gfCNCPoint3[3648] = {X 36.5946, Y 43.2362, Z -3.8333, A 0.000, B 0.000, C 0.000 }
gfCNCPoint3[3649] = {X 36.9340, Y 42.3177, Z -3.8333, A 0.000, B 0.000, C 0.000 }
gfCNCPoint3[3650] = {X 37.4786, Y 41.5040, Z -3.8333, A 0.000, B 0.000, C 0.000 }
gfCNCPoint3[3651] = {X 38.1984, Y 40.8401, Z -3.8333, A 0.000, B 0.000, C 0.000 }
gfCNCPoint3[3652] = {X 39.0535, Y 40.3629, Z -3.8333, A 0.000, B 0.000, C 0.000 }
gfCNCPoint3[3653] = {X 39.6603, Y 38.9339, Z -3.8333, A 0.000, B 0.000, C 0.000 }
gfCNCPoint3[3654] = {X 40.2151, Y 37.4838, Z -3.8333, A 0.000, B 0.000, C 0.000 }
gfCNCPoint3[3655] = {X 43.7985, Y 27.8628, Z -3.8333, A 0.000, B 0.000, C 0.000 }
gfCNCPoint3[3656] = {X 40.0500, Y 26.4667, Z -3.8333, A 0.000, B 0.000, C 0.000 }
gfCNCPoint3[3657] = {X 43.8734, Y 27.8908, Z -3.8333, A 0.000, B 0.000, C 0.000 }
gfCNCPoint3[3658] = {X 48.5582, Y 15.3126, Z -3.8333, A 0.000, B 0.000, C 0.000 }
gfCNCPoint3[3659] = {X 48.1610, Y 14.6012, Z -3.8333, A 0.000, B 0.000, C 0.000 }
gfCNCPoint3[3660] = {X 47.9131, Y 13.8250, Z -3.8333, A 0.000, B 0.000, C 0.000 }
gfCNCPoint3[3661] = {X 47.8244, Y 13.0151, Z -3.8333, A 0.000, B 0.000, C 0.000 }
gfCNCPoint3[3662] = {X 47.8242, Y 12.1868, Z -3.8333, A 0.000, B 0.000, C 0.000 }
gfCNCPoint3[3663] = {X 47.9265, Y 11.2789, Z -3.8333, A 0.000, B 0.000, C 0.000 }
gfCNCPoint3[3664] = {X 48.2283, Y 10.4166, Z -3.8333, A 0.000, B 0.000, C 0.000 }
gfCNCPoint3[3665] = {X 48.7144, Y 9.6430, Z -3.8333, A 0.000, B 0.000, C 0.000 }
gfCNCPoint3[3666] = {X 49.3604, Y 8.9969, Z -3.8333, A 0.000, B 0.000, C 0.000 }
gfCNCPoint3[3667] = {X 50.1340, Y 8.5109, Z -3.8333, A 0.000, B 0.000, C 0.000 }
gfCNCPoint3[3668] = {X 50.9963, Y 8.2091, Z -3.8333, A 0.000, B 0.000, C 0.000 }
gfCNCPoint3[3669] = {X 51.9042, Y 8.1068, Z -3.8333, A 0.000, B 0.000, C 0.000 }
gfCNCPoint3[3670] = {X 59.6221, Y 8.1068, Z -3.8333, A 0.000, B 0.000, C 0.000 }
gfCNCPoint3[3671] = {X 60.5300, Y 8.2091, Z -3.8333, A 0.000, B 0.000, C 0.000 }
gfCNCPoint3[3672] = {X 61.3924, Y 8.5109, Z -3.8333, A 0.000, B 0.000, C 0.000 }
gfCNCPoint3[3673] = {X 62.1660, Y 8.9969, Z -3.8333, A 0.000, B 0.000, C 0.000 }
gfCNCPoint3[3674] = {X 62.8120, Y 9.6430, Z -3.8333, A 0.000, B 0.000, C 0.000 }
gfCNCPoint3[3675] = {X 63.2981, Y 10.4166, Z -3.8333, A 0.000, B 0.000, C 0.000 }
gfCNCPoint3[3676] = {X 63.5998, Y 11.2789, Z -3.8333, A 0.000, B 0.000, C 0.000 }
gfCNCPoint3[3677] = {X 63.7021, Y 12.1868, Z -3.8333, A 0.000, B 0.000, C 0.000 }
gfCNCPoint3[3678] = {X 63.7021, Y 12.9781, Z -3.8333, A 0.000, B 0.000, C 0.000 }
gfCNCPoint3[3679] = {X 63.6148, Y 13.8178, Z -3.8333, A 0.000, B 0.000, C 0.000 }
gfCNCPoint3[3680] = {X 63.3565, Y 14.6215, Z -3.8333, A 0.000, B 0.000, C 0.000 }
gfCNCPoint3[3681] = {X 62.9383, Y 15.3549, Z -3.8333, A 0.000, B 0.000, C 0.000 }
gfCNCPoint3[3682] = {X 63.2010, Y 16.0481, Z -3.8333, A 0.000, B 0.000, C 0.000 }
gfCNCPoint3[3683] = {X 66.0153, Y 23.5156, Z -3.8333, A 0.000, B 0.000, C 0.000 }
gfCNCPoint3[3684] = {X 71.9853, Y 39.5865, Z -3.8333, A 0.000, B 0.000, C 0.000 }
gfCNCPoint3[3685] = {X 72.3281, Y 40.4487, Z -3.8333, A 0.000, B 0.000, C 0.000 }
gfCNCPoint3[3686] = {X 73.1522, Y 40.9150, Z -3.8333, A 0.000, B 0.000, C 0.000 }
gfCNCPoint3[3687] = {X 73.8466, Y 41.5587, Z -3.8333, A 0.000, B 0.000, C 0.000 }
gfCNCPoint3[3688] = {X 74.3739, Y 42.3451, Z -3.8333, A 0.000, B 0.000, C 0.000 }
gfCNCPoint3[3689] = {X 74.7058, Y 43.2319, Z -3.8333, A 0.000, B 0.000, C 0.000 }
gfCNCPoint3[3690] = {X 74.8243, Y 44.1714, Z -3.8333, A 0.000, B 0.000, C 0.000 }
gfCNCPoint3[3691] = {X 74.8245, Y 45.0000, Z -3.8333, A 0.000, B 0.000, C 0.000 }
gfCNCPoint3[3692] = {X 74.7222, Y 45.9079, Z -3.8333, A 0.000, B 0.000, C 0.000 }
gfCNCPoint3[3693] = {X 74.4204, Y 46.7702, Z -3.8333, A 0.000, B 0.000, C 0.000 }
gfCNCPoint3[3694] = {X 73.9343, Y 47.5438, Z -3.8333, A 0.000, B 0.000, C 0.000 }
gfCNCPoint3[3695] = {X 73.2883, Y 48.1899, Z -3.8333, A 0.000, B 0.000, C 0.000 }
gfCNCPoint3[3696] = {X 72.5147, Y 48.6760, Z -3.8333, A 0.000, B 0.000, C 0.000 }
gfCNCPoint3[3697] = {X 71.6523, Y 48.9777, Z -3.8333, A 0.000, B 0.000, C 0.000 }
gfCNCPoint3[3698] = {X 70.7445, Y 49.0800, Z -3.8333, A 0.000, B 0.000, C 0.000 }
gfCNCPoint3[3699] = {X 64.1851, Y 49.0800, Z -3.8333, A 0.000, B 0.000, C 0.000 }
gfCNCPoint3[3700] = {X 63.2772, Y 48.9777, Z -3.8333, A 0.000, B 0.000, C 0.000 }
gfCNCPoint3[3701] = {X 62.4149, Y 48.6760, Z -3.8333, A 0.000, B 0.000, C 0.000 }
gfCNCPoint3[3702] = {X 61.6413, Y 48.1899, Z -3.8333, A 0.000, B 0.000, C 0.000 }
gfCNCPoint3[3703] = {X 60.9953, Y 47.5438, Z -3.8333, A 0.000, B 0.000, C 0.000 }
gfCNCPoint3[3704] = {X 60.5092, Y 46.7702, Z -3.8333, A 0.000, B 0.000, C 0.000 }
gfCNCPoint3[3705] = {X 60.2074, Y 45.9079, Z -3.8333, A 0.000, B 0.000, C 0.000 }
gfCNCPoint3[3706] = {X 60.1051, Y 45.0000, Z -3.8333, A 0.000, B 0.000, C 0.000 }
gfCNCPoint3[3707] = {X 60.1051, Y 44.2086, Z -3.8333, A 0.000, B 0.000, C 0.000 }
gfCNCPoint3[3708] = {X 60.1954, Y 43.3580, Z -3.8333, A 0.000, B 0.000, C 0.000 }
gfCNCPoint3[3709] = {X 60.4611, Y 42.5449, Z -3.8333, A 0.000, B 0.000, C 0.000 }
gfCNCPoint3[3710] = {X 60.8905, Y 41.8050, Z -3.8333, A 0.000, B 0.000, C 0.000 }
gfCNCPoint3[3711] = {X 60.1748, Y 39.8492, Z -3.8333, A 0.000, B 0.000, C 0.000 }
gfCNCPoint3[3712] = {X 51.9103, Y 39.8492, Z -3.8333, A 0.000, B 0.000, C 0.000 }
gfCNCPoint3[3713] = {X 51.0690, Y 42.1092, Z -3.8333, A 0.000, B 0.000, C 0.000 }
gfCNCPoint3[3714] = {X 51.1306, Y 42.2115, Z -3.8333, A 0.000, B 0.000, C 0.000 }
gfCNCPoint3[3715] = {X 51.4141, Y 42.8332, Z -3.8333, A 0.000, B 0.000, C 0.000 }
gfCNCPoint3[3716] = {X 51.5898, Y 43.4936, Z -3.8333, A 0.000, B 0.000, C 0.000 }
gfCNCPoint3[3717] = {X 51.6528, Y 44.1740, Z -3.8333, A 0.000, B 0.000, C 0.000 }
gfCNCPoint3[3718] = {X 51.6529, Y 45.0000, Z -3.8333, A 0.000, B 0.000, C 0.000 }
gfCNCPoint3[3719] = {X 51.5506, Y 45.9079, Z -3.8333, A 0.000, B 0.000, C 0.000 }
gfCNCPoint3[3720] = {X 51.2489, Y 46.7702, Z -3.8333, A 0.000, B 0.000, C 0.000 }
gfCNCPoint3[3721] = {X 50.7628, Y 47.5438, Z -3.8333, A 0.000, B 0.000, C 0.000 }
gfCNCPoint3[3722] = {X 50.1168, Y 48.1899, Z -3.8333, A 0.000, B 0.000, C 0.000 }
gfCNCPoint3[3723] = {X 49.3432, Y 48.6760, Z -3.8333, A 0.000, B 0.000, C 0.000 }
gfCNCPoint3[3724] = {X 48.4808, Y 48.9777, Z -3.8333, A 0.000, B 0.000, C 0.000 }
gfCNCPoint3[3725] = {X 47.5729, Y 49.0800, Z -3.8333, A 0.000, B 0.000, C 0.000 }
gfCNCPoint3[3726] = {X 40.6393, Y 49.0800, Z -3.8333, A 0.000, B 0.000, C 0.000 }
gfCNCPoint3[3727] = {X 39.7314, Y 48.9777, Z -3.8333, A 0.000, B 0.000, C 0.000 }
gfCNCPoint3[3728] = {X 38.8691, Y 48.6760, Z -3.8333, A 0.000, B 0.000, C 0.000 }
gfCNCPoint3[3729] = {X 38.0955, Y 48.1899, Z -3.8333, A 0.000, B 0.000, C 0.000 }
gfCNCPoint3[3730] = {X 37.4494, Y 47.5438, Z -3.8333, A 0.000, B 0.000, C 0.000 }
gfCNCPoint3[3731] = {X 36.9633, Y 46.7702, Z -3.8333, A 0.000, B 0.000, C 0.000 }
gfCNCPoint3[3732] = {X 36.6616, Y 45.9079, Z -3.8333, A 0.000, B 0.000, C 0.000 }
gfCNCPoint3[3733] = {X 36.5593, Y 45.0000, Z -3.8333, A 0.000, B 0.000, C 0.000 }
gfCNCPoint3[3734] = {X 36.5593, Y 44.2086, Z -3.8333, A 0.000, B 0.000, C 0.000 }
gfCNCPoint3[3735] = {X 36.6737, Y 43.2478, Z -3.8333, A 0.000, B 0.000, C 0.000 }
gfCNCPoint3[3736] = {X 37.0110, Y 42.3409, Z -3.8333, A 0.000, B 0.000, C 0.000 }
gfCNCPoint3[3737] = {X 37.5522, Y 41.5388, Z -3.8333, A 0.000, B 0.000, C 0.000 }
gfCNCPoint3[3738] = {X 38.2670, Y 40.8866, Z -3.8333, A 0.000, B 0.000, C 0.000 }
gfCNCPoint3[3739] = {X 39.1152, Y 40.4209, Z -3.8333, A 0.000, B 0.000, C 0.000 }
gfCNCPoint3[3740] = {X 39.1265, Y 40.3955, Z -3.8333, A 0.000, B 0.000, C 0.000 }
gfCNCPoint3[3741] = {X 39.7345, Y 38.9638, Z -3.8333, A 0.000, B 0.000, C 0.000 }
gfCNCPoint3[3742] = {X 40.2904, Y 37.5110, Z -3.8333, A 0.000, B 0.000, C 0.000 }
gfCNCPoint3[3743] = {X 43.8734, Y 27.8908, Z -3.8333, A 0.000, B 0.000, C 0.000 }
gfCNCPoint3[3744] = {X 40.1250, Y 26.4946, Z -3.8333, A 0.000, B 0.000, C 0.000 }
gfCNCPoint3[3745] = {X 43.9484, Y 27.9187, Z -3.8333, A 0.000, B 0.000, C 0.000 }
gfCNCPoint3[3746] = {X 48.6479, Y 15.3010, Z -3.8333, A 0.000, B 0.000, C 0.000 }
gfCNCPoint3[3747] = {X 48.2407, Y 14.5838, Z -3.8333, A 0.000, B 0.000, C 0.000 }
gfCNCPoint3[3748] = {X 47.9892, Y 13.7983, Z -3.8333, A 0.000, B 0.000, C 0.000 }
gfCNCPoint3[3749] = {X 47.9042, Y 12.9779, Z -3.8333, A 0.000, B 0.000, C 0.000 }
gfCNCPoint3[3750] = {X 47.9042, Y 12.1868, Z -3.8333, A 0.000, B 0.000, C 0.000 }
gfCNCPoint3[3751] = {X 48.0045, Y 11.2967, Z -3.8333, A 0.000, B 0.000, C 0.000 }
gfCNCPoint3[3752] = {X 48.3003, Y 10.4513, Z -3.8333, A 0.000, B 0.000, C 0.000 }
gfCNCPoint3[3753] = {X 48.7769, Y 9.6929, Z -3.8333, A 0.000, B 0.000, C 0.000 }
gfCNCPoint3[3754] = {X 49.4103, Y 9.0595, Z -3.8333, A 0.000, B 0.000, C 0.000 }
gfCNCPoint3[3755] = {X 50.1687, Y 8.5829, Z -3.8333, A 0.000, B 0.000, C 0.000 }
gfCNCPoint3[3756] = {X 51.0141, Y 8.2871, Z -3.8333, A 0.000, B 0.000, C 0.000 }
gfCNCPoint3[3757] = {X 51.9042, Y 8.1868, Z -3.8333, A 0.000, B 0.000, C 0.000 }
gfCNCPoint3[3758] = {X 59.6221, Y 8.1868, Z -3.8333, A 0.000, B 0.000, C 0.000 }
gfCNCPoint3[3759] = {X 60.5122, Y 8.2871, Z -3.8333, A 0.000, B 0.000, C 0.000 }
gfCNCPoint3[3760] = {X 61.3577, Y 8.5829, Z -3.8333, A 0.000, B 0.000, C 0.000 }
gfCNCPoint3[3761] = {X 62.1161, Y 9.0595, Z -3.8333, A 0.000, B 0.000, C 0.000 }
gfCNCPoint3[3762] = {X 62.7495, Y 9.6929, Z -3.8333, A 0.000, B 0.000, C 0.000 }
gfCNCPoint3[3763] = {X 63.2260, Y 10.4513, Z -3.8333, A 0.000, B 0.000, C 0.000 }
gfCNCPoint3[3764] = {X 63.5218, Y 11.2967, Z -3.8333, A 0.000, B 0.000, C 0.000 }
gfCNCPoint3[3765] = {X 63.6221, Y 12.1868, Z -3.8333, A 0.000, B 0.000, C 0.000 }
gfCNCPoint3[3766] = {X 63.6219, Y 13.0192, Z -3.8333, A 0.000, B 0.000, C 0.000 }
gfCNCPoint3[3767] = {X 63.5277, Y 13.8420, Z -3.8333, A 0.000, B 0.000, C 0.000 }
gfCNCPoint3[3768] = {X 63.2660, Y 14.6278, Z -3.8333, A 0.000, B 0.000, C 0.000 }
gfCNCPoint3[3769] = {X 62.8482, Y 15.3429, Z -3.8333, A 0.000, B 0.000, C 0.000 }
gfCNCPoint3[3770] = {X 63.1261, Y 16.0764, Z -3.8333, A 0.000, B 0.000, C 0.000 }
gfCNCPoint3[3771] = {X 65.9404, Y 23.5436, Z -3.8333, A 0.000, B 0.000, C 0.000 }
gfCNCPoint3[3772] = {X 71.9107, Y 39.6152, Z -3.8333, A 0.000, B 0.000, C 0.000 }
gfCNCPoint3[3773] = {X 72.2611, Y 40.4966, Z -3.8333, A 0.000, B 0.000, C 0.000 }
gfCNCPoint3[3774] = {X 72.2790, Y 40.5149, Z -3.8333, A 0.000, B 0.000, C 0.000 }
gfCNCPoint3[3775] = {X 72.3450, Y 40.5429, Z -3.8333, A 0.000, B 0.000, C 0.000 }
gfCNCPoint3[3776] = {X 72.4104, Y 40.5722, Z -3.8333, A 0.000, B 0.000, C 0.000 }
gfCNCPoint3[3777] = {X 73.1900, Y 41.0435, Z -3.8333, A 0.000, B 0.000, C 0.000 }
gfCNCPoint3[3778] = {X 73.8428, Y 41.6790, Z -3.8333, A 0.000, B 0.000, C 0.000 }
gfCNCPoint3[3779] = {X 74.3349, Y 42.4457, Z -3.8333, A 0.000, B 0.000, C 0.000 }
gfCNCPoint3[3780] = {X 74.6407, Y 43.3038, Z -3.8333, A 0.000, B 0.000, C 0.000 }
gfCNCPoint3[3781] = {X 74.7445, Y 44.2089, Z -3.8333, A 0.000, B 0.000, C 0.000 }
gfCNCPoint3[3782] = {X 74.7445, Y 45.0000, Z -3.8333, A 0.000, B 0.000, C 0.000 }
gfCNCPoint3[3783] = {X 74.6442, Y 45.8901, Z -3.8333, A 0.000, B 0.000, C 0.000 }
gfCNCPoint3[3784] = {X 74.3483, Y 46.7355, Z -3.8333, A 0.000, B 0.000, C 0.000 }
gfCNCPoint3[3785] = {X 73.8718, Y 47.4940, Z -3.8333, A 0.000, B 0.000, C 0.000 }
gfCNCPoint3[3786] = {X 73.2384, Y 48.1273, Z -3.8333, A 0.000, B 0.000, C 0.000 }
gfCNCPoint3[3787] = {X 72.4800, Y 48.6039, Z -3.8333, A 0.000, B 0.000, C 0.000 }
gfCNCPoint3[3788] = {X 71.6345, Y 48.8997, Z -3.8333, A 0.000, B 0.000, C 0.000 }
gfCNCPoint3[3789] = {X 70.7445, Y 49.0000, Z -3.8333, A 0.000, B 0.000, C 0.000 }
gfCNCPoint3[3790] = {X 64.1851, Y 49.0000, Z -3.8333, A 0.000, B 0.000, C 0.000 }
gfCNCPoint3[3791] = {X 63.2951, Y 48.8997, Z -3.8333, A 0.000, B 0.000, C 0.000 }
gfCNCPoint3[3792] = {X 62.4496, Y 48.6039, Z -3.8333, A 0.000, B 0.000, C 0.000 }
gfCNCPoint3[3793] = {X 61.6912, Y 48.1273, Z -3.8333, A 0.000, B 0.000, C 0.000 }
gfCNCPoint3[3794] = {X 61.0578, Y 47.4940, Z -3.8333, A 0.000, B 0.000, C 0.000 }
gfCNCPoint3[3795] = {X 60.5813, Y 46.7355, Z -3.8333, A 0.000, B 0.000, C 0.000 }
gfCNCPoint3[3796] = {X 60.2854, Y 45.8901, Z -3.8333, A 0.000, B 0.000, C 0.000 }
gfCNCPoint3[3797] = {X 60.1851, Y 45.0000, Z -3.8333, A 0.000, B 0.000, C 0.000 }
gfCNCPoint3[3798] = {X 60.1855, Y 44.1538, Z -3.8333, A 0.000, B 0.000, C 0.000 }
gfCNCPoint3[3799] = {X 60.2746, Y 43.3674, Z -3.8333, A 0.000, B 0.000, C 0.000 }
gfCNCPoint3[3800] = {X 60.5168, Y 42.6140, Z -3.8333, A 0.000, B 0.000, C 0.000 }
gfCNCPoint3[3801] = {X 60.9025, Y 41.9231, Z -3.8333, A 0.000, B 0.000, C 0.000 }
gfCNCPoint3[3802] = {X 60.9805, Y 41.8180, Z -3.8333, A 0.000, B 0.000, C 0.000 }
gfCNCPoint3[3803] = {X 60.2307, Y 39.7692, Z -3.8333, A 0.000, B 0.000, C 0.000 }
gfCNCPoint3[3804] = {X 51.8423, Y 39.7692, Z -3.8333, A 0.000, B 0.000, C 0.000 }
gfCNCPoint3[3805] = {X 51.8423, Y 39.8027, Z -3.8333, A 0.000, B 0.000, C 0.000 }
gfCNCPoint3[3806] = {X 50.9806, Y 42.1175, Z -3.8333, A 0.000, B 0.000, C 0.000 }
gfCNCPoint3[3807] = {X 51.0724, Y 42.2713, Z -3.8333, A 0.000, B 0.000, C 0.000 }
gfCNCPoint3[3808] = {X 51.3478, Y 42.8858, Z -3.8333, A 0.000, B 0.000, C 0.000 }
gfCNCPoint3[3809] = {X 51.5163, Y 43.5378, Z -3.8333, A 0.000, B 0.000, C 0.000 }
gfCNCPoint3[3810] = {X 51.5729, Y 44.2089, Z -3.8333, A 0.000, B 0.000, C 0.000 }
gfCNCPoint3[3811] = {X 51.5729, Y 45.0000, Z -3.8333, A 0.000, B 0.000, C 0.000 }
gfCNCPoint3[3812] = {X 51.4726, Y 45.8901, Z -3.8333, A 0.000, B 0.000, C 0.000 }
gfCNCPoint3[3813] = {X 51.1768, Y 46.7355, Z -3.8333, A 0.000, B 0.000, C 0.000 }
gfCNCPoint3[3814] = {X 50.7003, Y 47.4940, Z -3.8333, A 0.000, B 0.000, C 0.000 }
gfCNCPoint3[3815] = {X 50.0669, Y 48.1273, Z -3.8333, A 0.000, B 0.000, C 0.000 }
gfCNCPoint3[3816] = {X 49.3085, Y 48.6039, Z -3.8333, A 0.000, B 0.000, C 0.000 }
gfCNCPoint3[3817] = {X 48.4630, Y 48.8997, Z -3.8333, A 0.000, B 0.000, C 0.000 }
gfCNCPoint3[3818] = {X 47.5729, Y 49.0000, Z -3.8333, A 0.000, B 0.000, C 0.000 }
gfCNCPoint3[3819] = {X 40.6393, Y 49.0000, Z -3.8333, A 0.000, B 0.000, C 0.000 }
gfCNCPoint3[3820] = {X 39.7492, Y 48.8997, Z -3.8333, A 0.000, B 0.000, C 0.000 }
gfCNCPoint3[3821] = {X 38.9038, Y 48.6039, Z -3.8333, A 0.000, B 0.000, C 0.000 }
gfCNCPoint3[3822] = {X 38.1453, Y 48.1273, Z -3.8333, A 0.000, B 0.000, C 0.000 }
gfCNCPoint3[3823] = {X 37.5120, Y 47.4940, Z -3.8333, A 0.000, B 0.000, C 0.000 }
gfCNCPoint3[3824] = {X 37.0354, Y 46.7355, Z -3.8333, A 0.000, B 0.000, C 0.000 }
gfCNCPoint3[3825] = {X 36.7396, Y 45.8901, Z -3.8333, A 0.000, B 0.000, C 0.000 }
gfCNCPoint3[3826] = {X 36.6393, Y 45.0000, Z -3.8333, A 0.000, B 0.000, C 0.000 }
gfCNCPoint3[3827] = {X 36.6397, Y 44.1538, Z -3.8333, A 0.000, B 0.000, C 0.000 }
gfCNCPoint3[3828] = {X 36.7564, Y 43.2482, Z -3.8333, A 0.000, B 0.000, C 0.000 }
gfCNCPoint3[3829] = {X 37.0754, Y 42.3926, Z -3.8333, A 0.000, B 0.000, C 0.000 }
gfCNCPoint3[3830] = {X 37.5801, Y 41.6317, Z -3.8333, A 0.000, B 0.000, C 0.000 }
gfCNCPoint3[3831] = {X 38.2442, Y 41.0051, Z -3.8333, A 0.000, B 0.000, C 0.000 }
gfCNCPoint3[3832] = {X 39.0332, Y 40.5454, Z -3.8333, A 0.000, B 0.000, C 0.000 }
gfCNCPoint3[3833] = {X 39.0861, Y 40.5226, Z -3.8333, A 0.000, B 0.000, C 0.000 }
gfCNCPoint3[3834] = {X 39.1394, Y 40.5006, Z -3.8333, A 0.000, B 0.000, C 0.000 }
gfCNCPoint3[3835] = {X 39.1684, Y 40.4818, Z -3.8333, A 0.000, B 0.000, C 0.000 }
gfCNCPoint3[3836] = {X 39.1882, Y 40.4536, Z -3.8333, A 0.000, B 0.000, C 0.000 }
gfCNCPoint3[3837] = {X 39.2132, Y 40.3974, Z -3.8333, A 0.000, B 0.000, C 0.000 }
gfCNCPoint3[3838] = {X 39.2382, Y 40.3412, Z -3.8333, A 0.000, B 0.000, C 0.000 }
gfCNCPoint3[3839] = {X 39.8265, Y 38.9496, Z -3.8333, A 0.000, B 0.000, C 0.000 }
gfCNCPoint3[3840] = {X 40.3656, Y 37.5383, Z -3.8333, A 0.000, B 0.000, C 0.000 }
gfCNCPoint3[3841] = {X 43.9484, Y 27.9187, Z -3.8333, A 0.000, B 0.000, C 0.000 }
gfCNCPoint3[3842] = {X 40.1250, Y 26.4946, Z -3.8333, A 0.000, B 0.000, C 0.000 }
gfCNCPoint3[3843] = {X 40.1250, Y 26.4946, Z -0.8333, A 0.000, B 0.000, C 0.000 }
gfCNCPoint3[3844] = {X 40.1250, Y 26.4946, Z 11.0000, A 0.000, B 0.000, C 0.000 }
gfCNCPoint3[3845] = {X 79.0230, Y 28.5918, Z 11.0000, A 0.000, B 0.000, C 0.000 }
gfCNCPoint3[3846] = {X 79.0230, Y 28.5918, Z -0.8333, A 0.000, B 0.000, C 0.000 }
gfCNCPoint3[3847] = {X 79.0230, Y 28.5918, Z -3.8333, A 0.000, B 0.000, C 0.000 }
gfCNCPoint3[3848] = {X 83.1030, Y 28.5918, Z -3.8333, A 0.000, B 0.000, C 0.000 }
gfCNCPoint3[3849] = {X 83.1028, Y 16.2743, Z -3.8333, A 0.000, B 0.000, C 0.000 }
gfCNCPoint3[3850] = {X 82.4642, Y 15.6032, Z -3.8333, A 0.000, B 0.000, C 0.000 }
gfCNCPoint3[3851] = {X 81.9834, Y 14.8113, Z -3.8333, A 0.000, B 0.000, C 0.000 }
gfCNCPoint3[3852] = {X 81.6824, Y 13.9352, Z -3.8333, A 0.000, B 0.000, C 0.000 }
gfCNCPoint3[3853] = {X 81.5752, Y 13.0150, Z -3.8333, A 0.000, B 0.000, C 0.000 }
gfCNCPoint3[3854] = {X 81.5751, Y 12.1868, Z -3.8333, A 0.000, B 0.000, C 0.000 }
gfCNCPoint3[3855] = {X 81.6834, Y 11.2255, Z -3.8333, A 0.000, B 0.000, C 0.000 }
gfCNCPoint3[3856] = {X 82.0029, Y 10.3124, Z -3.8333, A 0.000, B 0.000, C 0.000 }
gfCNCPoint3[3857] = {X 82.5176, Y 9.4933, Z -3.8333, A 0.000, B 0.000, C 0.000 }
gfCNCPoint3[3858] = {X 83.2016, Y 8.8093, Z -3.8333, A 0.000, B 0.000, C 0.000 }
gfCNCPoint3[3859] = {X 84.0207, Y 8.2946, Z -3.8333, A 0.000, B 0.000, C 0.000 }
gfCNCPoint3[3860] = {X 84.9338, Y 7.9751, Z -3.8333, A 0.000, B 0.000, C 0.000 }
gfCNCPoint3[3861] = {X 85.8951, Y 7.8668, Z -3.8333, A 0.000, B 0.000, C 0.000 }
gfCNCPoint3[3862] = {X 94.0497, Y 7.8668, Z -3.8333, A 0.000, B 0.000, C 0.000 }
gfCNCPoint3[3863] = {X 95.0110, Y 7.9751, Z -3.8333, A 0.000, B 0.000, C 0.000 }
gfCNCPoint3[3864] = {X 95.9240, Y 8.2946, Z -3.8333, A 0.000, B 0.000, C 0.000 }
gfCNCPoint3[3865] = {X 96.7431, Y 8.8093, Z -3.8333, A 0.000, B 0.000, C 0.000 }
gfCNCPoint3[3866] = {X 97.4272, Y 9.4933, Z -3.8333, A 0.000, B 0.000, C 0.000 }
gfCNCPoint3[3867] = {X 97.9419, Y 10.3124, Z -3.8333, A 0.000, B 0.000, C 0.000 }
gfCNCPoint3[3868] = {X 98.2614, Y 11.2255, Z -3.8333, A 0.000, B 0.000, C 0.000 }
gfCNCPoint3[3869] = {X 98.3697, Y 12.1868, Z -3.8333, A 0.000, B 0.000, C 0.000 }
gfCNCPoint3[3870] = {X 98.3697, Y 12.9782, Z -3.8333, A 0.000, B 0.000, C 0.000 }
gfCNCPoint3[3871] = {X 98.2967, Y 13.7681, Z -3.8333, A 0.000, B 0.000, C 0.000 }
gfCNCPoint3[3872] = {X 98.0804, Y 14.5314, Z -3.8333, A 0.000, B 0.000, C 0.000 }
gfCNCPoint3[3873] = {X 97.7283, Y 15.2423, Z -3.8333, A 0.000, B 0.000, C 0.000 }
gfCNCPoint3[3874] = {X 101.8779, Y 25.5293, Z -3.8333, A 0.000, B 0.000, C 0.000 }
gfCNCPoint3[3875] = {X 106.0166, Y 15.2216, Z -3.8333, A 0.000, B 0.000, C 0.000 }
gfCNCPoint3[3876] = {X 105.6762, Y 14.5287, Z -3.8333, A 0.000, B 0.000, C 0.000 }
gfCNCPoint3[3877] = {X 105.4645, Y 13.7862, Z -3.8333, A 0.000, B 0.000, C 0.000 }
gfCNCPoint3[3878] = {X 105.3885, Y 13.0179, Z -3.8333, A 0.000, B 0.000, C 0.000 }
gfCNCPoint3[3879] = {X 105.3883, Y 12.1868, Z -3.8333, A 0.000, B 0.000, C 0.000 }
gfCNCPoint3[3880] = {X 105.4966, Y 11.2255, Z -3.8333, A 0.000, B 0.000, C 0.000 }
gfCNCPoint3[3881] = {X 105.8161, Y 10.3124, Z -3.8333, A 0.000, B 0.000, C 0.000 }
gfCNCPoint3[3882] = {X 106.3308, Y 9.4933, Z -3.8333, A 0.000, B 0.000, C 0.000 }
gfCNCPoint3[3883] = {X 107.0148, Y 8.8093, Z -3.8333, A 0.000, B 0.000, C 0.000 }
gfCNCPoint3[3884] = {X 107.8339, Y 8.2946, Z -3.8333, A 0.000, B 0.000, C 0.000 }
gfCNCPoint3[3885] = {X 108.7470, Y 7.9751, Z -3.8333, A 0.000, B 0.000, C 0.000 }
gfCNCPoint3[3886] = {X 109.7083, Y 7.8668, Z -3.8333, A 0.000, B 0.000, C 0.000 }
gfCNCPoint3[3887] = {X 117.7916, Y 7.8668, Z -3.8333, A 0.000, B 0.000, C 0.000 }
gfCNCPoint3[3888] = {X 118.7529, Y 7.9751, Z -3.8333, A 0.000, B 0.000, C 0.000 }
gfCNCPoint3[3889] = {X 119.6660, Y 8.2946, Z -3.8333, A 0.000, B 0.000, C 0.000 }
gfCNCPoint3[3890] = {X 120.4851, Y 8.8093, Z -3.8333, A 0.000, B 0.000, C 0.000 }
gfCNCPoint3[3891] = {X 121.1691, Y 9.4933, Z -3.8333, A 0.000, B 0.000, C 0.000 }
gfCNCPoint3[3892] = {X 121.6838, Y 10.3124, Z -3.8333, A 0.000, B 0.000, C 0.000 }
gfCNCPoint3[3893] = {X 122.0033, Y 11.2255, Z -3.8333, A 0.000, B 0.000, C 0.000 }
gfCNCPoint3[3894] = {X 122.1116, Y 12.1868, Z -3.8333, A 0.000, B 0.000, C 0.000 }
gfCNCPoint3[3895] = {X 122.1116, Y 12.9782, Z -3.8333, A 0.000, B 0.000, C 0.000 }
gfCNCPoint3[3896] = {X 122.0103, Y 13.9078, Z -3.8333, A 0.000, B 0.000, C 0.000 }
gfCNCPoint3[3897] = {X 121.7114, Y 14.7940, Z -3.8333, A 0.000, B 0.000, C 0.000 }
gfCNCPoint3[3898] = {X 121.2287, Y 15.5950, Z -3.8333, A 0.000, B 0.000, C 0.000 }
gfCNCPoint3[3899] = {X 120.5850, Y 16.2734, Z -3.8333, A 0.000, B 0.000, C 0.000 }
gfCNCPoint3[3900] = {X 120.5838, Y 40.9140, Z -3.8333, A 0.000, B 0.000, C 0.000 }
gfCNCPoint3[3901] = {X 120.6221, Y 40.9452, Z -3.8333, A 0.000, B 0.000, C 0.000 }
gfCNCPoint3[3902] = {X 121.2455, Y 41.6140, Z -3.8333, A 0.000, B 0.000, C 0.000 }
gfCNCPoint3[3903] = {X 121.7142, Y 42.3990, Z -3.8333, A 0.000, B 0.000, C 0.000 }
gfCNCPoint3[3904] = {X 122.0072, Y 43.2651, Z -3.8333, A 0.000, B 0.000, C 0.000 }
gfCNCPoint3[3905] = {X 122.1114, Y 44.1734, Z -3.8333, A 0.000, B 0.000, C 0.000 }
gfCNCPoint3[3906] = {X 122.1116, Y 45.0000, Z -3.8333, A 0.000, B 0.000, C 0.000 }
gfCNCPoint3[3907] = {X 122.0033, Y 45.9613, Z -3.8333, A 0.000, B 0.000, C 0.000 }
gfCNCPoint3[3908] = {X 121.6838, Y 46.8744, Z -3.8333, A 0.000, B 0.000, C 0.000 }
gfCNCPoint3[3909] = {X 121.1691, Y 47.6935, Z -3.8333, A 0.000, B 0.000, C 0.000 }
gfCNCPoint3[3910] = {X 120.4851, Y 48.3775, Z -3.8333, A 0.000, B 0.000, C 0.000 }
gfCNCPoint3[3911] = {X 119.6660, Y 48.8922, Z -3.8333, A 0.000, B 0.000, C 0.000 }
gfCNCPoint3[3912] = {X 118.7529, Y 49.2117, Z -3.8333, A 0.000, B 0.000, C 0.000 }
gfCNCPoint3[3913] = {X 117.7916, Y 49.3200, Z -3.8333, A 0.000, B 0.000, C 0.000 }
gfCNCPoint3[3914] = {X 111.9185, Y 49.3200, Z -3.8333, A 0.000, B 0.000, C 0.000 }
gfCNCPoint3[3915] = {X 110.9619, Y 49.2128, Z -3.8333, A 0.000, B 0.000, C 0.000 }
gfCNCPoint3[3916] = {X 110.0529, Y 48.8964, Z -3.8333, A 0.000, B 0.000, C 0.000 }
gfCNCPoint3[3917] = {X 109.2365, Y 48.3866, Z -3.8333, A 0.000, B 0.000, C 0.000 }
gfCNCPoint3[3918] = {X 108.5532, Y 47.7087, Z -3.8333, A 0.000, B 0.000, C 0.000 }
gfCNCPoint3[3919] = {X 108.0369, Y 46.8963, Z -3.8333, A 0.000, B 0.000, C 0.000 }
gfCNCPoint3[3920] = {X 107.7134, Y 45.9898, Z -3.8333, A 0.000, B 0.000, C 0.000 }
gfCNCPoint3[3921] = {X 107.5986, Y 45.0341, Z -3.8333, A 0.000, B 0.000, C 0.000 }
gfCNCPoint3[3922] = {X 107.5985, Y 44.1793, Z -3.8333, A 0.000, B 0.000, C 0.000 }
gfCNCPoint3[3923] = {X 107.6342, Y 43.6358, Z -3.8333, A 0.000, B 0.000, C 0.000 }
gfCNCPoint3[3924] = {X 107.7408, Y 43.1017, Z -3.8333, A 0.000, B 0.000, C 0.000 }
gfCNCPoint3[3925] = {X 107.9078, Y 42.6067, Z -3.8333, A 0.000, B 0.000, C 0.000 }
gfCNCPoint3[3926] = {X 108.1357, Y 42.1366, Z -3.8333, A 0.000, B 0.000, C 0.000 }
gfCNCPoint3[3927] = {X 108.5865, Y 41.4649, Z -3.8333, A 0.000, B 0.000, C 0.000 }
gfCNCPoint3[3928] = {X 109.1263, Y 40.8623, Z -3.8333, A 0.000, B 0.000, C 0.000 }
gfCNCPoint3[3929] = {X 109.1262, Y 39.2953, Z -3.8333, A 0.000, B 0.000, C 0.000 }
gfCNCPoint3[3930] = {X 106.1118, Y 46.6615, Z -3.8333, A 0.000, B 0.000, C 0.000 }
gfCNCPoint3[3931] = {X 105.7417, Y 47.3611, Z -3.8333, A 0.000, B 0.000, C 0.000 }
gfCNCPoint3[3932] = {X 105.2502, Y 47.9815, Z -3.8333, A 0.000, B 0.000, C 0.000 }
gfCNCPoint3[3933] = {X 104.6538, Y 48.5018, Z -3.8333, A 0.000, B 0.000, C 0.000 }
gfCNCPoint3[3934] = {X 103.9724, Y 48.9046, Z -3.8333, A 0.000, B 0.000, C 0.000 }
gfCNCPoint3[3935] = {X 103.0287, Y 49.2242, Z -3.8333, A 0.000, B 0.000, C 0.000 }
gfCNCPoint3[3936] = {X 102.0368, Y 49.3191, Z -3.8333, A 0.000, B 0.000, C 0.000 }
gfCNCPoint3[3937] = {X 101.0496, Y 49.1842, Z -3.8333, A 0.000, B 0.000, C 0.000 }
gfCNCPoint3[3938] = {X 100.1195, Y 48.8268, Z -3.8333, A 0.000, B 0.000, C 0.000 }
gfCNCPoint3[3939] = {X 99.2961, Y 48.2657, Z -3.8333, A 0.000, B 0.000, C 0.000 }
gfCNCPoint3[3940] = {X 98.6231, Y 47.5309, Z -3.8333, A 0.000, B 0.000, C 0.000 }
gfCNCPoint3[3941] = {X 98.1363, Y 46.6615, Z -3.8333, A 0.000, B 0.000, C 0.000 }
gfCNCPoint3[3942] = {X 95.1307, Y 39.3109, Z -3.8333, A 0.000, B 0.000, C 0.000 }
gfCNCPoint3[3943] = {X 95.1308, Y 40.9052, Z -3.8333, A 0.000, B 0.000, C 0.000 }
gfCNCPoint3[3944] = {X 95.6590, Y 41.4465, Z -3.8333, A 0.000, B 0.000, C 0.000 }
gfCNCPoint3[3945] = {X 96.0868, Y 42.0702, Z -3.8333, A 0.000, B 0.000, C 0.000 }
gfCNCPoint3[3946] = {X 96.3310, Y 42.5736, Z -3.8333, A 0.000, B 0.000, C 0.000 }
gfCNCPoint3[3947] = {X 96.5094, Y 43.1039, Z -3.8333, A 0.000, B 0.000, C 0.000 }
gfCNCPoint3[3948] = {X 96.6189, Y 43.6504, Z -3.8333, A 0.000, B 0.000, C 0.000 }
gfCNCPoint3[3949] = {X 96.6585, Y 44.2064, Z -3.8333, A 0.000, B 0.000, C 0.000 }
gfCNCPoint3[3950] = {X 96.6583, Y 45.0415, Z -3.8333, A 0.000, B 0.000, C 0.000 }
gfCNCPoint3[3951] = {X 96.5422, Y 45.9960, Z -3.8333, A 0.000, B 0.000, C 0.000 }
gfCNCPoint3[3952] = {X 96.2178, Y 46.9011, Z -3.8333, A 0.000, B 0.000, C 0.000 }
gfCNCPoint3[3953] = {X 95.7012, Y 47.7120, Z -3.8333, A 0.000, B 0.000, C 0.000 }
gfCNCPoint3[3954] = {X 95.0181, Y 48.3886, Z -3.8333, A 0.000, B 0.000, C 0.000 }
gfCNCPoint3[3955] = {X 94.2022, Y 48.8973, Z -3.8333, A 0.000, B 0.000, C 0.000 }
gfCNCPoint3[3956] = {X 93.2940, Y 49.2130, Z -3.8333, A 0.000, B 0.000, C 0.000 }
gfCNCPoint3[3957] = {X 92.3385, Y 49.3200, Z -3.8333, A 0.000, B 0.000, C 0.000 }
gfCNCPoint3[3958] = {X 85.8951, Y 49.3200, Z -3.8333, A 0.000, B 0.000, C 0.000 }
gfCNCPoint3[3959] = {X 84.9387, Y 49.2128, Z -3.8333, A 0.000, B 0.000, C 0.000 }
gfCNCPoint3[3960] = {X 84.0297, Y 48.8965, Z -3.8333, A 0.000, B 0.000, C 0.000 }
gfCNCPoint3[3961] = {X 83.2134, Y 48.3869, Z -3.8333, A 0.000, B 0.000, C 0.000 }
gfCNCPoint3[3962] = {X 82.5301, Y 47.7091, Z -3.8333, A 0.000, B 0.000, C 0.000 }
gfCNCPoint3[3963] = {X 82.0138, Y 46.8970, Z -3.8333, A 0.000, B 0.000, C 0.000 }
gfCNCPoint3[3964] = {X 81.6902, Y 45.9906, Z -3.8333, A 0.000, B 0.000, C 0.000 }
gfCNCPoint3[3965] = {X 81.5752, Y 45.0351, Z -3.8333, A 0.000, B 0.000, C 0.000 }
gfCNCPoint3[3966] = {X 81.5751, Y 44.2070, Z -3.8333, A 0.000, B 0.000, C 0.000 }
gfCNCPoint3[3967] = {X 81.6805, Y 43.2777, Z -3.8333, A 0.000, B 0.000, C 0.000 }
gfCNCPoint3[3968] = {X 81.9808, Y 42.3921, Z -3.8333, A 0.000, B 0.000, C 0.000 }
gfCNCPoint3[3969] = {X 82.4624, Y 41.5904, Z -3.8333, A 0.000, B 0.000, C 0.000 }
gfCNCPoint3[3970] = {X 83.1031, Y 40.9092, Z -3.8333, A 0.000, B 0.000, C 0.000 }
gfCNCPoint3[3971] = {X 83.1030, Y 28.5918, Z -3.8333, A 0.000, B 0.000, C 0.000 }
gfCNCPoint3[3972] = {X 79.1030, Y 28.5918, Z -3.8333, A 0.000, B 0.000, C 0.000 }
gfCNCPoint3[3973] = {X 83.1830, Y 28.5918, Z -3.8333, A 0.000, B 0.000, C 0.000 }
gfCNCPoint3[3974] = {X 83.1828, Y 16.2370, Z -3.8333, A 0.000, B 0.000, C 0.000 }
gfCNCPoint3[3975] = {X 82.5446, Y 15.5765, Z -3.8333, A 0.000, B 0.000, C 0.000 }
gfCNCPoint3[3976] = {X 82.0637, Y 14.7941, Z -3.8333, A 0.000, B 0.000, C 0.000 }
gfCNCPoint3[3977] = {X 81.7625, Y 13.9264, Z -3.8333, A 0.000, B 0.000, C 0.000 }
gfCNCPoint3[3978] = {X 81.6552, Y 13.0143, Z -3.8333, A 0.000, B 0.000, C 0.000 }
gfCNCPoint3[3979] = {X 81.6551, Y 12.1868, Z -3.8333, A 0.000, B 0.000, C 0.000 }
gfCNCPoint3[3980] = {X 81.7614, Y 11.2433, Z -3.8333, A 0.000, B 0.000, C 0.000 }
gfCNCPoint3[3981] = {X 82.0750, Y 10.3472, Z -3.8333, A 0.000, B 0.000, C 0.000 }
gfCNCPoint3[3982] = {X 82.5801, Y 9.5432, Z -3.8333, A 0.000, B 0.000, C 0.000 }
gfCNCPoint3[3983] = {X 83.2515, Y 8.8719, Z -3.8333, A 0.000, B 0.000, C 0.000 }
gfCNCPoint3[3984] = {X 84.0554, Y 8.3667, Z -3.8333, A 0.000, B 0.000, C 0.000 }
gfCNCPoint3[3985] = {X 84.9516, Y 8.0531, Z -3.8333, A 0.000, B 0.000, C 0.000 }
gfCNCPoint3[3986] = {X 85.8951, Y 7.9468, Z -3.8333, A 0.000, B 0.000, C 0.000 }
gfCNCPoint3[3987] = {X 94.0497, Y 7.9468, Z -3.8333, A 0.000, B 0.000, C 0.000 }
gfCNCPoint3[3988] = {X 94.9932, Y 8.0531, Z -3.8333, A 0.000, B 0.000, C 0.000 }
gfCNCPoint3[3989] = {X 95.8893, Y 8.3667, Z -3.8333, A 0.000, B 0.000, C 0.000 }
gfCNCPoint3[3990] = {X 96.6933, Y 8.8718, Z -3.8333, A 0.000, B 0.000, C 0.000 }
gfCNCPoint3[3991] = {X 97.3646, Y 9.5432, Z -3.8333, A 0.000, B 0.000, C 0.000 }
gfCNCPoint3[3992] = {X 97.8698, Y 10.3471, Z -3.8333, A 0.000, B 0.000, C 0.000 }
gfCNCPoint3[3993] = {X 98.1834, Y 11.2433, Z -3.8333, A 0.000, B 0.000, C 0.000 }
gfCNCPoint3[3994] = {X 98.2897, Y 12.1868, Z -3.8333, A 0.000, B 0.000, C 0.000 }
gfCNCPoint3[3995] = {X 98.2897, Y 12.9782, Z -3.8333, A 0.000, B 0.000, C 0.000 }
gfCNCPoint3[3996] = {X 98.2155, Y 13.7667, Z -3.8333, A 0.000, B 0.000, C 0.000 }
gfCNCPoint3[3997] = {X 97.9960, Y 14.5276, Z -3.8333, A 0.000, B 0.000, C 0.000 }
gfCNCPoint3[3998] = {X 97.6389, Y 15.2345, Z -3.8333, A 0.000, B 0.000, C 0.000 }
gfCNCPoint3[3999] = {X 101.8778, Y 25.7430, Z -3.8333, A 0.000, B 0.000, C 0.000 }
gfCNCPoint3[4000] = {X 101.9521, Y 25.5591, Z -3.8333, A 0.000, B 0.000, C 0.000 }
gfCNCPoint3[4001] = {X 106.1058, Y 15.2141, Z -3.8333, A 0.000, B 0.000, C 0.000 }
gfCNCPoint3[4002] = {X 105.7605, Y 14.5247, Z -3.8333, A 0.000, B 0.000, C 0.000 }
gfCNCPoint3[4003] = {X 105.5456, Y 13.7843, Z -3.8333, A 0.000, B 0.000, C 0.000 }
gfCNCPoint3[4004] = {X 105.4685, Y 13.0172, Z -3.8333, A 0.000, B 0.000, C 0.000 }
gfCNCPoint3[4005] = {X 105.4683, Y 12.1868, Z -3.8333, A 0.000, B 0.000, C 0.000 }
gfCNCPoint3[4006] = {X 105.5746, Y 11.2433, Z -3.8333, A 0.000, B 0.000, C 0.000 }
gfCNCPoint3[4007] = {X 105.8882, Y 10.3471, Z -3.8333, A 0.000, B 0.000, C 0.000 }
gfCNCPoint3[4008] = {X 106.3933, Y 9.5432, Z -3.8333, A 0.000, B 0.000, C 0.000 }
gfCNCPoint3[4009] = {X 107.0647, Y 8.8718, Z -3.8333, A 0.000, B 0.000, C 0.000 }
gfCNCPoint3[4010] = {X 107.8686, Y 8.3667, Z -3.8333, A 0.000, B 0.000, C 0.000 }
gfCNCPoint3[4011] = {X 108.7648, Y 8.0531, Z -3.8333, A 0.000, B 0.000, C 0.000 }
gfCNCPoint3[4012] = {X 109.7083, Y 7.9468, Z -3.8333, A 0.000, B 0.000, C 0.000 }
gfCNCPoint3[4013] = {X 117.7916, Y 7.9468, Z -3.8333, A 0.000, B 0.000, C 0.000 }
gfCNCPoint3[4014] = {X 118.7351, Y 8.0531, Z -3.8333, A 0.000, B 0.000, C 0.000 }
gfCNCPoint3[4015] = {X 119.6312, Y 8.3667, Z -3.8333, A 0.000, B 0.000, C 0.000 }
gfCNCPoint3[4016] = {X 120.4352, Y 8.8718, Z -3.8333, A 0.000, B 0.000, C 0.000 }
gfCNCPoint3[4017] = {X 121.1065, Y 9.5432, Z -3.8333, A 0.000, B 0.000, C 0.000 }
gfCNCPoint3[4018] = {X 121.6117, Y 10.3471, Z -3.8333, A 0.000, B 0.000, C 0.000 }
gfCNCPoint3[4019] = {X 121.9253, Y 11.2433, Z -3.8333, A 0.000, B 0.000, C 0.000 }
gfCNCPoint3[4020] = {X 122.0316, Y 12.1868, Z -3.8333, A 0.000, B 0.000, C 0.000 }
gfCNCPoint3[4021] = {X 122.0316, Y 12.9782, Z -3.8333, A 0.000, B 0.000, C 0.000 }
gfCNCPoint3[4022] = {X 121.9302, Y 13.8996, Z -3.8333, A 0.000, B 0.000, C 0.000 }
gfCNCPoint3[4023] = {X 121.6310, Y 14.7771, Z -3.8333, A 0.000, B 0.000, C 0.000 }
gfCNCPoint3[4024] = {X 121.1482, Y 15.5685, Z -3.8333, A 0.000, B 0.000, C 0.000 }
gfCNCPoint3[4025] = {X 120.5050, Y 16.2361, Z -3.8333, A 0.000, B 0.000, C 0.000 }
gfCNCPoint3[4026] = {X 120.5038, Y 40.9520, Z -3.8333, A 0.000, B 0.000, C 0.000 }
gfCNCPoint3[4027] = {X 120.5706, Y 41.0065, Z -3.8333, A 0.000, B 0.000, C 0.000 }
gfCNCPoint3[4028] = {X 121.1821, Y 41.6628, Z -3.8333, A 0.000, B 0.000, C 0.000 }
gfCNCPoint3[4029] = {X 121.6418, Y 42.4331, Z -3.8333, A 0.000, B 0.000, C 0.000 }
gfCNCPoint3[4030] = {X 121.9292, Y 43.2828, Z -3.8333, A 0.000, B 0.000, C 0.000 }
gfCNCPoint3[4031] = {X 122.0314, Y 44.1740, Z -3.8333, A 0.000, B 0.000, C 0.000 }
gfCNCPoint3[4032] = {X 122.0316, Y 45.0000, Z -3.8333, A 0.000, B 0.000, C 0.000 }
gfCNCPoint3[4033] = {X 121.9253, Y 45.9435, Z -3.8333, A 0.000, B 0.000, C 0.000 }
gfCNCPoint3[4034] = {X 121.6117, Y 46.8397, Z -3.8333, A 0.000, B 0.000, C 0.000 }
gfCNCPoint3[4035] = {X 121.1065, Y 47.6436, Z -3.8333, A 0.000, B 0.000, C 0.000 }
gfCNCPoint3[4036] = {X 120.4352, Y 48.3150, Z -3.8333, A 0.000, B 0.000, C 0.000 }
gfCNCPoint3[4037] = {X 119.6312, Y 48.8201, Z -3.8333, A 0.000, B 0.000, C 0.000 }
gfCNCPoint3[4038] = {X 118.7351, Y 49.1337, Z -3.8333, A 0.000, B 0.000, C 0.000 }
gfCNCPoint3[4039] = {X 117.7916, Y 49.2400, Z -3.8333, A 0.000, B 0.000, C 0.000 }
gfCNCPoint3[4040] = {X 111.9185, Y 49.2400, Z -3.8333, A 0.000, B 0.000, C 0.000 }
gfCNCPoint3[4041] = {X 110.9797, Y 49.1348, Z -3.8333, A 0.000, B 0.000, C 0.000 }
gfCNCPoint3[4042] = {X 110.0874, Y 48.8242, Z -3.8333, A 0.000, B 0.000, C 0.000 }
gfCNCPoint3[4043] = {X 109.2861, Y 48.3239, Z -3.8333, A 0.000, B 0.000, C 0.000 }
gfCNCPoint3[4044] = {X 108.6155, Y 47.6585, Z -3.8333, A 0.000, B 0.000, C 0.000 }
gfCNCPoint3[4045] = {X 108.1088, Y 46.8612, Z -3.8333, A 0.000, B 0.000, C 0.000 }
gfCNCPoint3[4046] = {X 107.7913, Y 45.9714, Z -3.8333, A 0.000, B 0.000, C 0.000 }
gfCNCPoint3[4047] = {X 107.6786, Y 45.0335, Z -3.8333, A 0.000, B 0.000, C 0.000 }
gfCNCPoint3[4048] = {X 107.6785, Y 44.1793, Z -3.8333, A 0.000, B 0.000, C 0.000 }
gfCNCPoint3[4049] = {X 107.7135, Y 43.6463, Z -3.8333, A 0.000, B 0.000, C 0.000 }
gfCNCPoint3[4050] = {X 107.8180, Y 43.1225, Z -3.8333, A 0.000, B 0.000, C 0.000 }
gfCNCPoint3[4051] = {X 107.9818, Y 42.6370, Z -3.8333, A 0.000, B 0.000, C 0.000 }
gfCNCPoint3[4052] = {X 108.2053, Y 42.1760, Z -3.8333, A 0.000, B 0.000, C 0.000 }
gfCNCPoint3[4053] = {X 108.6602, Y 41.5005, Z -3.8333, A 0.000, B 0.000, C 0.000 }
gfCNCPoint3[4054] = {X 109.2063, Y 40.8962, Z -3.8333, A 0.000, B 0.000, C 0.000 }
gfCNCPoint3[4055] = {X 109.2061, Y 39.1629, Z -3.8333, A 0.000, B 0.000, C 0.000 }
gfCNCPoint3[4056] = {X 109.0939, Y 39.1629, Z -3.8333, A 0.000, B 0.000, C 0.000 }
gfCNCPoint3[4057] = {X 106.0379, Y 46.6307, Z -3.8333, A 0.000, B 0.000, C 0.000 }
gfCNCPoint3[4058] = {X 105.6747, Y 47.3174, Z -3.8333, A 0.000, B 0.000, C 0.000 }
gfCNCPoint3[4059] = {X 105.1923, Y 47.9263, Z -3.8333, A 0.000, B 0.000, C 0.000 }
gfCNCPoint3[4060] = {X 104.6069, Y 48.4370, Z -3.8333, A 0.000, B 0.000, C 0.000 }
gfCNCPoint3[4061] = {X 103.9382, Y 48.8323, Z -3.8333, A 0.000, B 0.000, C 0.000 }
gfCNCPoint3[4062] = {X 103.0119, Y 49.1460, Z -3.8333, A 0.000, B 0.000, C 0.000 }
gfCNCPoint3[4063] = {X 102.0384, Y 49.2391, Z -3.8333, A 0.000, B 0.000, C 0.000 }
gfCNCPoint3[4064] = {X 101.0695, Y 49.1068, Z -3.8333, A 0.000, B 0.000, C 0.000 }
gfCNCPoint3[4065] = {X 100.1566, Y 48.7559, Z -3.8333, A 0.000, B 0.000, C 0.000 }
gfCNCPoint3[4066] = {X 99.3484, Y 48.2052, Z -3.8333, A 0.000, B 0.000, C 0.000 }
gfCNCPoint3[4067] = {X 98.6879, Y 47.4840, Z -3.8333, A 0.000, B 0.000, C 0.000 }
gfCNCPoint3[4068] = {X 98.2102, Y 46.6307, Z -3.8333, A 0.000, B 0.000, C 0.000 }
gfCNCPoint3[4069] = {X 95.0507, Y 38.9038, Z -3.8333, A 0.000, B 0.000, C 0.000 }
gfCNCPoint3[4070] = {X 95.0508, Y 40.9421, Z -3.8333, A 0.000, B 0.000, C 0.000 }
gfCNCPoint3[4071] = {X 95.5855, Y 41.4832, Z -3.8333, A 0.000, B 0.000, C 0.000 }
gfCNCPoint3[4072] = {X 96.0172, Y 42.1096, Z -3.8333, A 0.000, B 0.000, C 0.000 }
gfCNCPoint3[4073] = {X 96.2570, Y 42.6039, Z -3.8333, A 0.000, B 0.000, C 0.000 }
gfCNCPoint3[4074] = {X 96.4322, Y 43.1246, Z -3.8333, A 0.000, B 0.000, C 0.000 }
gfCNCPoint3[4075] = {X 96.5397, Y 43.6612, Z -3.8333, A 0.000, B 0.000, C 0.000 }
gfCNCPoint3[4076] = {X 96.5785, Y 44.2070, Z -3.8333, A 0.000, B 0.000, C 0.000 }
gfCNCPoint3[4077] = {X 96.5783, Y 45.0408, Z -3.8333, A 0.000, B 0.000, C 0.000 }
gfCNCPoint3[4078] = {X 96.4643, Y 45.9775, Z -3.8333, A 0.000, B 0.000, C 0.000 }
gfCNCPoint3[4079] = {X 96.1459, Y 46.8659, Z -3.8333, A 0.000, B 0.000, C 0.000 }
gfCNCPoint3[4080] = {X 95.6389, Y 47.6618, Z -3.8333, A 0.000, B 0.000, C 0.000 }
gfCNCPoint3[4081] = {X 94.9685, Y 48.3258, Z -3.8333, A 0.000, B 0.000, C 0.000 }
gfCNCPoint3[4082] = {X 94.1677, Y 48.8251, Z -3.8333, A 0.000, B 0.000, C 0.000 }
gfCNCPoint3[4083] = {X 93.2764, Y 49.1350, Z -3.8333, A 0.000, B 0.000, C 0.000 }
gfCNCPoint3[4084] = {X 92.3385, Y 49.2400, Z -3.8333, A 0.000, B 0.000, C 0.000 }
gfCNCPoint3[4085] = {X 85.8951, Y 49.2400, Z -3.8333, A 0.000, B 0.000, C 0.000 }
gfCNCPoint3[4086] = {X 84.9564, Y 49.1348, Z -3.8333, A 0.000, B 0.000, C 0.000 }
gfCNCPoint3[4087] = {X 84.0643, Y 48.8244, Z -3.8333, A 0.000, B 0.000, C 0.000 }
gfCNCPoint3[4088] = {X 83.2631, Y 48.3242, Z -3.8333, A 0.000, B 0.000, C 0.000 }
gfCNCPoint3[4089] = {X 82.5924, Y 47.6590, Z -3.8333, A 0.000, B 0.000, C 0.000 }
gfCNCPoint3[4090] = {X 82.0857, Y 46.8618, Z -3.8333, A 0.000, B 0.000, C 0.000 }
gfCNCPoint3[4091] = {X 81.7681, Y 45.9723, Z -3.8333, A 0.000, B 0.000, C 0.000 }
gfCNCPoint3[4092] = {X 81.6552, Y 45.0345, Z -3.8333, A 0.000, B 0.000, C 0.000 }
gfCNCPoint3[4093] = {X 81.6551, Y 44.2074, Z -3.8333, A 0.000, B 0.000, C 0.000 }
gfCNCPoint3[4094] = {X 81.7606, Y 43.2863, Z -3.8333, A 0.000, B 0.000, C 0.000 }
gfCNCPoint3[4095] = {X 82.0612, Y 42.4091, Z -3.8333, A 0.000, B 0.000, C 0.000 }
gfCNCPoint3[4096] = {X 82.5428, Y 41.6168, Z -3.8333, A 0.000, B 0.000, C 0.000 }
gfCNCPoint3[4097] = {X 83.1831, Y 40.9462, Z -3.8333, A 0.000, B 0.000, C 0.000 }
gfCNCPoint3[4098] = {X 83.1830, Y 28.5918, Z -3.8333, A 0.000, B 0.000, C 0.000 }
gfCNCPoint3[4099] = {X 79.1830, Y 28.5918, Z -3.8333, A 0.000, B 0.000, C 0.000 }
gfCNCPoint3[4100] = {X 83.2630, Y 28.5918, Z -3.8333, A 0.000, B 0.000, C 0.000 }
gfCNCPoint3[4101] = {X 83.2628, Y 16.1993, Z -3.8333, A 0.000, B 0.000, C 0.000 }
gfCNCPoint3[4102] = {X 82.6251, Y 15.5496, Z -3.8333, A 0.000, B 0.000, C 0.000 }
gfCNCPoint3[4103] = {X 82.1440, Y 14.7767, Z -3.8333, A 0.000, B 0.000, C 0.000 }
gfCNCPoint3[4104] = {X 81.8426, Y 13.9176, Z -3.8333, A 0.000, B 0.000, C 0.000 }
gfCNCPoint3[4105] = {X 81.7352, Y 13.0136, Z -3.8333, A 0.000, B 0.000, C 0.000 }
gfCNCPoint3[4106] = {X 81.7351, Y 12.1868, Z -3.8333, A 0.000, B 0.000, C 0.000 }
gfCNCPoint3[4107] = {X 81.8394, Y 11.2611, Z -3.8333, A 0.000, B 0.000, C 0.000 }
gfCNCPoint3[4108] = {X 82.1470, Y 10.3819, Z -3.8333, A 0.000, B 0.000, C 0.000 }
gfCNCPoint3[4109] = {X 82.6427, Y 9.5931, Z -3.8333, A 0.000, B 0.000, C 0.000 }
gfCNCPoint3[4110] = {X 83.3014, Y 8.9344, Z -3.8333, A 0.000, B 0.000, C 0.000 }
gfCNCPoint3[4111] = {X 84.0901, Y 8.4388, Z -3.8333, A 0.000, B 0.000, C 0.000 }
gfCNCPoint3[4112] = {X 84.9694, Y 8.1311, Z -3.8333, A 0.000, B 0.000, C 0.000 }
gfCNCPoint3[4113] = {X 85.8951, Y 8.0268, Z -3.8333, A 0.000, B 0.000, C 0.000 }
gfCNCPoint3[4114] = {X 94.0497, Y 8.0268, Z -3.8333, A 0.000, B 0.000, C 0.000 }
gfCNCPoint3[4115] = {X 94.9754, Y 8.1311, Z -3.8333, A 0.000, B 0.000, C 0.000 }
gfCNCPoint3[4116] = {X 95.8546, Y 8.4388, Z -3.8333, A 0.000, B 0.000, C 0.000 }
gfCNCPoint3[4117] = {X 96.6434, Y 8.9344, Z -3.8333, A 0.000, B 0.000, C 0.000 }
gfCNCPoint3[4118] = {X 97.3021, Y 9.5931, Z -3.8333, A 0.000, B 0.000, C 0.000 }
gfCNCPoint3[4119] = {X 97.7977, Y 10.3819, Z -3.8333, A 0.000, B 0.000, C 0.000 }
gfCNCPoint3[4120] = {X 98.1054, Y 11.2611, Z -3.8333, A 0.000, B 0.000, C 0.000 }
gfCNCPoint3[4121] = {X 98.2097, Y 12.1868, Z -3.8333, A 0.000, B 0.000, C 0.000 }
gfCNCPoint3[4122] = {X 98.2097, Y 12.9782, Z -3.8333, A 0.000, B 0.000, C 0.000 }
gfCNCPoint3[4123] = {X 98.1343, Y 13.7660, Z -3.8333, A 0.000, B 0.000, C 0.000 }
gfCNCPoint3[4124] = {X 97.9112, Y 14.5254, Z -3.8333, A 0.000, B 0.000, C 0.000 }
gfCNCPoint3[4125] = {X 97.5482, Y 15.2288, Z -3.8333, A 0.000, B 0.000, C 0.000 }
gfCNCPoint3[4126] = {X 101.8773, Y 25.9556, Z -3.8333, A 0.000, B 0.000, C 0.000 }
gfCNCPoint3[4127] = {X 101.9782, Y 25.7088, Z -3.8333, A 0.000, B 0.000, C 0.000 }
gfCNCPoint3[4128] = {X 106.1952, Y 15.2061, Z -3.8333, A 0.000, B 0.000, C 0.000 }
gfCNCPoint3[4129] = {X 105.8448, Y 14.5206, Z -3.8333, A 0.000, B 0.000, C 0.000 }
gfCNCPoint3[4130] = {X 105.6268, Y 13.7823, Z -3.8333, A 0.000, B 0.000, C 0.000 }
gfCNCPoint3[4131] = {X 105.5485, Y 13.0164, Z -3.8333, A 0.000, B 0.000, C 0.000 }
gfCNCPoint3[4132] = {X 105.5483, Y 12.1868, Z -3.8333, A 0.000, B 0.000, C 0.000 }
gfCNCPoint3[4133] = {X 105.6526, Y 11.2611, Z -3.8333, A 0.000, B 0.000, C 0.000 }
gfCNCPoint3[4134] = {X 105.9602, Y 10.3819, Z -3.8333, A 0.000, B 0.000, C 0.000 }
gfCNCPoint3[4135] = {X 106.4559, Y 9.5931, Z -3.8333, A 0.000, B 0.000, C 0.000 }
gfCNCPoint3[4136] = {X 107.1146, Y 8.9344, Z -3.8333, A 0.000, B 0.000, C 0.000 }
gfCNCPoint3[4137] = {X 107.9033, Y 8.4388, Z -3.8333, A 0.000, B 0.000, C 0.000 }
gfCNCPoint3[4138] = {X 108.7826, Y 8.1311, Z -3.8333, A 0.000, B 0.000, C 0.000 }
gfCNCPoint3[4139] = {X 109.7083, Y 8.0268, Z -3.8333, A 0.000, B 0.000, C 0.000 }
gfCNCPoint3[4140] = {X 117.7916, Y 8.0268, Z -3.8333, A 0.000, B 0.000, C 0.000 }
gfCNCPoint3[4141] = {X 118.7173, Y 8.1311, Z -3.8333, A 0.000, B 0.000, C 0.000 }
gfCNCPoint3[4142] = {X 119.5965, Y 8.4388, Z -3.8333, A 0.000, B 0.000, C 0.000 }
gfCNCPoint3[4143] = {X 120.3853, Y 8.9344, Z -3.8333, A 0.000, B 0.000, C 0.000 }
gfCNCPoint3[4144] = {X 121.0440, Y 9.5931, Z -3.8333, A 0.000, B 0.000, C 0.000 }
gfCNCPoint3[4145] = {X 121.5396, Y 10.3819, Z -3.8333, A 0.000, B 0.000, C 0.000 }
gfCNCPoint3[4146] = {X 121.8473, Y 11.2611, Z -3.8333, A 0.000, B 0.000, C 0.000 }
gfCNCPoint3[4147] = {X 121.9516, Y 12.1868, Z -3.8333, A 0.000, B 0.000, C 0.000 }
gfCNCPoint3[4148] = {X 121.9516, Y 12.9782, Z -3.8333, A 0.000, B 0.000, C 0.000 }
gfCNCPoint3[4149] = {X 121.8501, Y 13.8914, Z -3.8333, A 0.000, B 0.000, C 0.000 }
gfCNCPoint3[4150] = {X 121.5506, Y 14.7600, Z -3.8333, A 0.000, B 0.000, C 0.000 }
gfCNCPoint3[4151] = {X 121.0677, Y 15.5417, Z -3.8333, A 0.000, B 0.000, C 0.000 }
gfCNCPoint3[4152] = {X 120.4250, Y 16.1984, Z -3.8333, A 0.000, B 0.000, C 0.000 }
gfCNCPoint3[4153] = {X 120.4237, Y 40.9900, Z -3.8333, A 0.000, B 0.000, C 0.000 }
gfCNCPoint3[4154] = {X 120.5190, Y 41.0677, Z -3.8333, A 0.000, B 0.000, C 0.000 }
gfCNCPoint3[4155] = {X 121.1186, Y 41.7116, Z -3.8333, A 0.000, B 0.000, C 0.000 }
gfCNCPoint3[4156] = {X 121.5694, Y 42.4671, Z -3.8333, A 0.000, B 0.000, C 0.000 }
gfCNCPoint3[4157] = {X 121.8512, Y 43.3006, Z -3.8333, A 0.000, B 0.000, C 0.000 }
gfCNCPoint3[4158] = {X 121.9514, Y 44.1747, Z -3.8333, A 0.000, B 0.000, C 0.000 }
gfCNCPoint3[4159] = {X 121.9516, Y 45.0000, Z -3.8333, A 0.000, B 0.000, C 0.000 }
gfCNCPoint3[4160] = {X 121.8473, Y 45.9257, Z -3.8333, A 0.000, B 0.000, C 0.000 }
gfCNCPoint3[4161] = {X 121.5396, Y 46.8050, Z -3.8333, A 0.000, B 0.000, C 0.000 }
gfCNCPoint3[4162] = {X 121.0440, Y 47.5937, Z -3.8333, A 0.000, B 0.000, C 0.000 }
gfCNCPoint3[4163] = {X 120.3853, Y 48.2524, Z -3.8333, A 0.000, B 0.000, C 0.000 }
gfCNCPoint3[4164] = {X 119.5965, Y 48.7480, Z -3.8333, A 0.000, B 0.000, C 0.000 }
gfCNCPoint3[4165] = {X 118.7173, Y 49.0557, Z -3.8333, A 0.000, B 0.000, C 0.000 }
gfCNCPoint3[4166] = {X 117.7916, Y 49.1600, Z -3.8333, A 0.000, B 0.000, C 0.000 }
gfCNCPoint3[4167] = {X 111.9185, Y 49.1600, Z -3.8333, A 0.000, B 0.000, C 0.000 }
gfCNCPoint3[4168] = {X 110.9974, Y 49.0567, Z -3.8333, A 0.000, B 0.000, C 0.000 }
gfCNCPoint3[4169] = {X 110.1220, Y 48.7521, Z -3.8333, A 0.000, B 0.000, C 0.000 }
gfCNCPoint3[4170] = {X 109.3358, Y 48.2612, Z -3.8333, A 0.000, B 0.000, C 0.000 }
gfCNCPoint3[4171] = {X 108.6778, Y 47.6084, Z -3.8333, A 0.000, B 0.000, C 0.000 }
gfCNCPoint3[4172] = {X 108.1807, Y 46.8261, Z -3.8333, A 0.000, B 0.000, C 0.000 }
gfCNCPoint3[4173] = {X 107.8691, Y 45.9531, Z -3.8333, A 0.000, B 0.000, C 0.000 }
gfCNCPoint3[4174] = {X 107.7586, Y 45.0328, Z -3.8333, A 0.000, B 0.000, C 0.000 }
gfCNCPoint3[4175] = {X 107.7585, Y 44.1793, Z -3.8333, A 0.000, B 0.000, C 0.000 }
gfCNCPoint3[4176] = {X 107.7928, Y 43.6568, Z -3.8333, A 0.000, B 0.000, C 0.000 }
gfCNCPoint3[4177] = {X 107.8953, Y 43.1432, Z -3.8333, A 0.000, B 0.000, C 0.000 }
gfCNCPoint3[4178] = {X 108.0559, Y 42.6673, Z -3.8333, A 0.000, B 0.000, C 0.000 }
gfCNCPoint3[4179] = {X 108.2750, Y 42.2153, Z -3.8333, A 0.000, B 0.000, C 0.000 }
gfCNCPoint3[4180] = {X 108.7339, Y 41.5361, Z -3.8333, A 0.000, B 0.000, C 0.000 }
gfCNCPoint3[4181] = {X 109.2863, Y 40.9305, Z -3.8333, A 0.000, B 0.000, C 0.000 }
gfCNCPoint3[4182] = {X 109.2861, Y 39.0829, Z -3.8333, A 0.000, B 0.000, C 0.000 }
gfCNCPoint3[4183] = {X 109.0402, Y 39.0829, Z -3.8333, A 0.000, B 0.000, C 0.000 }
gfCNCPoint3[4184] = {X 105.9641, Y 46.5999, Z -3.8333, A 0.000, B 0.000, C 0.000 }
gfCNCPoint3[4185] = {X 105.6077, Y 47.2737, Z -3.8333, A 0.000, B 0.000, C 0.000 }
gfCNCPoint3[4186] = {X 105.1344, Y 47.8711, Z -3.8333, A 0.000, B 0.000, C 0.000 }
gfCNCPoint3[4187] = {X 104.5601, Y 48.3721, Z -3.8333, A 0.000, B 0.000, C 0.000 }
gfCNCPoint3[4188] = {X 103.9040, Y 48.7600, Z -3.8333, A 0.000, B 0.000, C 0.000 }
gfCNCPoint3[4189] = {X 102.9952, Y 49.0678, Z -3.8333, A 0.000, B 0.000, C 0.000 }
gfCNCPoint3[4190] = {X 102.0400, Y 49.1592, Z -3.8333, A 0.000, B 0.000, C 0.000 }
gfCNCPoint3[4191] = {X 101.0894, Y 49.0293, Z -3.8333, A 0.000, B 0.000, C 0.000 }
gfCNCPoint3[4192] = {X 100.1937, Y 48.6850, Z -3.8333, A 0.000, B 0.000, C 0.000 }
gfCNCPoint3[4193] = {X 99.4008, Y 48.1448, Z -3.8333, A 0.000, B 0.000, C 0.000 }
gfCNCPoint3[4194] = {X 98.7527, Y 47.4372, Z -3.8333, A 0.000, B 0.000, C 0.000 }
gfCNCPoint3[4195] = {X 98.2840, Y 46.5999, Z -3.8333, A 0.000, B 0.000, C 0.000 }
gfCNCPoint3[4196] = {X 94.9707, Y 38.4967, Z -3.8333, A 0.000, B 0.000, C 0.000 }
gfCNCPoint3[4197] = {X 94.9708, Y 40.9793, Z -3.8333, A 0.000, B 0.000, C 0.000 }
gfCNCPoint3[4198] = {X 95.5121, Y 41.5200, Z -3.8333, A 0.000, B 0.000, C 0.000 }
gfCNCPoint3[4199] = {X 95.9475, Y 42.1490, Z -3.8333, A 0.000, B 0.000, C 0.000 }
gfCNCPoint3[4200] = {X 96.1829, Y 42.6342, Z -3.8333, A 0.000, B 0.000, C 0.000 }
gfCNCPoint3[4201] = {X 96.3549, Y 43.1452, Z -3.8333, A 0.000, B 0.000, C 0.000 }
gfCNCPoint3[4202] = {X 96.4604, Y 43.6719, Z -3.8333, A 0.000, B 0.000, C 0.000 }
gfCNCPoint3[4203] = {X 96.4985, Y 44.2076, Z -3.8333, A 0.000, B 0.000, C 0.000 }
gfCNCPoint3[4204] = {X 96.4983, Y 45.0400, Z -3.8333, A 0.000, B 0.000, C 0.000 }
gfCNCPoint3[4205] = {X 96.3865, Y 45.9591, Z -3.8333, A 0.000, B 0.000, C 0.000 }
gfCNCPoint3[4206] = {X 96.0741, Y 46.8306, Z -3.8333, A 0.000, B 0.000, C 0.000 }
gfCNCPoint3[4207] = {X 95.5767, Y 47.6115, Z -3.8333, A 0.000, B 0.000, C 0.000 }
gfCNCPoint3[4208] = {X 94.9188, Y 48.2631, Z -3.8333, A 0.000, B 0.000, C 0.000 }
gfCNCPoint3[4209] = {X 94.1332, Y 48.7530, Z -3.8333, A 0.000, B 0.000, C 0.000 }
gfCNCPoint3[4210] = {X 93.2587, Y 49.0570, Z -3.8333, A 0.000, B 0.000, C 0.000 }
gfCNCPoint3[4211] = {X 92.3385, Y 49.1600, Z -3.8333, A 0.000, B 0.000, C 0.000 }
gfCNCPoint3[4212] = {X 85.8951, Y 49.1600, Z -3.8333, A 0.000, B 0.000, C 0.000 }
gfCNCPoint3[4213] = {X 84.9741, Y 49.0568, Z -3.8333, A 0.000, B 0.000, C 0.000 }
gfCNCPoint3[4214] = {X 84.0988, Y 48.7522, Z -3.8333, A 0.000, B 0.000, C 0.000 }
gfCNCPoint3[4215] = {X 83.3127, Y 48.2614, Z -3.8333, A 0.000, B 0.000, C 0.000 }
gfCNCPoint3[4216] = {X 82.6547, Y 47.6088, Z -3.8333, A 0.000, B 0.000, C 0.000 }
gfCNCPoint3[4217] = {X 82.1576, Y 46.8267, Z -3.8333, A 0.000, B 0.000, C 0.000 }
gfCNCPoint3[4218] = {X 81.8459, Y 45.9539, Z -3.8333, A 0.000, B 0.000, C 0.000 }
gfCNCPoint3[4219] = {X 81.7352, Y 45.0338, Z -3.8333, A 0.000, B 0.000, C 0.000 }
gfCNCPoint3[4220] = {X 81.7351, Y 44.2079, Z -3.8333, A 0.000, B 0.000, C 0.000 }
gfCNCPoint3[4221] = {X 81.8407, Y 43.2948, Z -3.8333, A 0.000, B 0.000, C 0.000 }
gfCNCPoint3[4222] = {X 82.1415, Y 42.4263, Z -3.8333, A 0.000, B 0.000, C 0.000 }
gfCNCPoint3[4223] = {X 82.6233, Y 41.6435, Z -3.8333, A 0.000, B 0.000, C 0.000 }
gfCNCPoint3[4224] = {X 83.2631, Y 40.9836, Z -3.8333, A 0.000, B 0.000, C 0.000 }
gfCNCPoint3[4225] = {X 83.2630, Y 28.5918, Z -3.8333, A 0.000, B 0.000, C 0.000 }
gfCNCPoint3[4226] = {X 79.2630, Y 28.5918, Z -3.8333, A 0.000, B 0.000, C 0.000 }
gfCNCPoint3[4227] = {X 83.3430, Y 28.5918, Z -3.8333, A 0.000, B 0.000, C 0.000 }
gfCNCPoint3[4228] = {X 83.3428, Y 16.1612, Z -3.8333, A 0.000, B 0.000, C 0.000 }
gfCNCPoint3[4229] = {X 82.7056, Y 15.5224, Z -3.8333, A 0.000, B 0.000, C 0.000 }
gfCNCPoint3[4230] = {X 82.2244, Y 14.7591, Z -3.8333, A 0.000, B 0.000, C 0.000 }
gfCNCPoint3[4231] = {X 81.9227, Y 13.9088, Z -3.8333, A 0.000, B 0.000, C 0.000 }
gfCNCPoint3[4232] = {X 81.8152, Y 13.0129, Z -3.8333, A 0.000, B 0.000, C 0.000 }
gfCNCPoint3[4233] = {X 81.8151, Y 12.1868, Z -3.8333, A 0.000, B 0.000, C 0.000 }
gfCNCPoint3[4234] = {X 81.9174, Y 11.2789, Z -3.8333, A 0.000, B 0.000, C 0.000 }
gfCNCPoint3[4235] = {X 82.2191, Y 10.4166, Z -3.8333, A 0.000, B 0.000, C 0.000 }
gfCNCPoint3[4236] = {X 82.7052, Y 9.6430, Z -3.8333, A 0.000, B 0.000, C 0.000 }
gfCNCPoint3[4237] = {X 83.3512, Y 8.9969, Z -3.8333, A 0.000, B 0.000, C 0.000 }
gfCNCPoint3[4238] = {X 84.1248, Y 8.5109, Z -3.8333, A 0.000, B 0.000, C 0.000 }
gfCNCPoint3[4239] = {X 84.9872, Y 8.2091, Z -3.8333, A 0.000, B 0.000, C 0.000 }
gfCNCPoint3[4240] = {X 85.8951, Y 8.1068, Z -3.8333, A 0.000, B 0.000, C 0.000 }
gfCNCPoint3[4241] = {X 94.0497, Y 8.1068, Z -3.8333, A 0.000, B 0.000, C 0.000 }
gfCNCPoint3[4242] = {X 94.9576, Y 8.2091, Z -3.8333, A 0.000, B 0.000, C 0.000 }
gfCNCPoint3[4243] = {X 95.8199, Y 8.5109, Z -3.8333, A 0.000, B 0.000, C 0.000 }
gfCNCPoint3[4244] = {X 96.5935, Y 8.9969, Z -3.8333, A 0.000, B 0.000, C 0.000 }
gfCNCPoint3[4245] = {X 97.2395, Y 9.6430, Z -3.8333, A 0.000, B 0.000, C 0.000 }
gfCNCPoint3[4246] = {X 97.7256, Y 10.4166, Z -3.8333, A 0.000, B 0.000, C 0.000 }
gfCNCPoint3[4247] = {X 98.0274, Y 11.2789, Z -3.8333, A 0.000, B 0.000, C 0.000 }
gfCNCPoint3[4248] = {X 98.1297, Y 12.1868, Z -3.8333, A 0.000, B 0.000, C 0.000 }
gfCNCPoint3[4249] = {X 98.1297, Y 12.9781, Z -3.8333, A 0.000, B 0.000, C 0.000 }
gfCNCPoint3[4250] = {X 98.0631, Y 13.7121, Z -3.8333, A 0.000, B 0.000, C 0.000 }
gfCNCPoint3[4251] = {X 97.8656, Y 14.4221, Z -3.8333, A 0.000, B 0.000, C 0.000 }
gfCNCPoint3[4252] = {X 97.5435, Y 15.0850, Z -3.8333, A 0.000, B 0.000, C 0.000 }
gfCNCPoint3[4253] = {X 97.4972, Y 15.1600, Z -3.8333, A 0.000, B 0.000, C 0.000 }
gfCNCPoint3[4254] = {X 97.4492, Y 15.2341, Z -3.8333, A 0.000, B 0.000, C 0.000 }
gfCNCPoint3[4255] = {X 97.4851, Y 15.2810, Z -3.8333, A 0.000, B 0.000, C 0.000 }
gfCNCPoint3[4256] = {X 101.8768, Y 26.1683, Z -3.8333, A 0.000, B 0.000, C 0.000 }
gfCNCPoint3[4257] = {X 102.0523, Y 25.7388, Z -3.8333, A 0.000, B 0.000, C 0.000 }
gfCNCPoint3[4258] = {X 106.2848, Y 15.1976, Z -3.8333, A 0.000, B 0.000, C 0.000 }
gfCNCPoint3[4259] = {X 106.2414, Y 15.1292, Z -3.8333, A 0.000, B 0.000, C 0.000 }
gfCNCPoint3[4260] = {X 106.1994, Y 15.0599, Z -3.8333, A 0.000, B 0.000, C 0.000 }
gfCNCPoint3[4261] = {X 105.8899, Y 14.4156, Z -3.8333, A 0.000, B 0.000, C 0.000 }
gfCNCPoint3[4262] = {X 105.6976, Y 13.7271, Z -3.8333, A 0.000, B 0.000, C 0.000 }
gfCNCPoint3[4263] = {X 105.6285, Y 13.0157, Z -3.8333, A 0.000, B 0.000, C 0.000 }
gfCNCPoint3[4264] = {X 105.6283, Y 12.1868, Z -3.8333, A 0.000, B 0.000, C 0.000 }
gfCNCPoint3[4265] = {X 105.7306, Y 11.2789, Z -3.8333, A 0.000, B 0.000, C 0.000 }
gfCNCPoint3[4266] = {X 106.0323, Y 10.4166, Z -3.8333, A 0.000, B 0.000, C 0.000 }
gfCNCPoint3[4267] = {X 106.5184, Y 9.6430, Z -3.8333, A 0.000, B 0.000, C 0.000 }
gfCNCPoint3[4268] = {X 107.1644, Y 8.9969, Z -3.8333, A 0.000, B 0.000, C 0.000 }
gfCNCPoint3[4269] = {X 107.9380, Y 8.5109, Z -3.8333, A 0.000, B 0.000, C 0.000 }
gfCNCPoint3[4270] = {X 108.8004, Y 8.2091, Z -3.8333, A 0.000, B 0.000, C 0.000 }
gfCNCPoint3[4271] = {X 109.7083, Y 8.1068, Z -3.8333, A 0.000, B 0.000, C 0.000 }
gfCNCPoint3[4272] = {X 117.7916, Y 8.1068, Z -3.8333, A 0.000, B 0.000, C 0.000 }
gfCNCPoint3[4273] = {X 118.6995, Y 8.2091, Z -3.8333, A 0.000, B 0.000, C 0.000 }
gfCNCPoint3[4274] = {X 119.5618, Y 8.5109, Z -3.8333, A 0.000, B 0.000, C 0.000 }
gfCNCPoint3[4275] = {X 120.3354, Y 8.9969, Z -3.8333, A 0.000, B 0.000, C 0.000 }
gfCNCPoint3[4276] = {X 120.9814, Y 9.6430, Z -3.8333, A 0.000, B 0.000, C 0.000 }
gfCNCPoint3[4277] = {X 121.4675, Y 10.4166, Z -3.8333, A 0.000, B 0.000, C 0.000 }
gfCNCPoint3[4278] = {X 121.7693, Y 11.2789, Z -3.8333, A 0.000, B 0.000, C 0.000 }
gfCNCPoint3[4279] = {X 121.8716, Y 12.1868, Z -3.8333, A 0.000, B 0.000, C 0.000 }
gfCNCPoint3[4280] = {X 121.8716, Y 12.9781, Z -3.8333, A 0.000, B 0.000, C 0.000 }
gfCNCPoint3[4281] = {X 121.7699, Y 13.8830, Z -3.8333, A 0.000, B 0.000, C 0.000 }
gfCNCPoint3[4282] = {X 121.4702, Y 14.7428, Z -3.8333, A 0.000, B 0.000, C 0.000 }
gfCNCPoint3[4283] = {X 120.9872, Y 15.5147, Z -3.8333, A 0.000, B 0.000, C 0.000 }
gfCNCPoint3[4284] = {X 120.3450, Y 16.1602, Z -3.8333, A 0.000, B 0.000, C 0.000 }
gfCNCPoint3[4285] = {X 120.3437, Y 41.0280, Z -3.8333, A 0.000, B 0.000, C 0.000 }
gfCNCPoint3[4286] = {X 120.4675, Y 41.1289, Z -3.8333, A 0.000, B 0.000, C 0.000 }
gfCNCPoint3[4287] = {X 121.0552, Y 41.7603, Z -3.8333, A 0.000, B 0.000, C 0.000 }
gfCNCPoint3[4288] = {X 121.4970, Y 42.5012, Z -3.8333, A 0.000, B 0.000, C 0.000 }
gfCNCPoint3[4289] = {X 121.7732, Y 43.3184, Z -3.8333, A 0.000, B 0.000, C 0.000 }
gfCNCPoint3[4290] = {X 121.8714, Y 44.1754, Z -3.8333, A 0.000, B 0.000, C 0.000 }
gfCNCPoint3[4291] = {X 121.8716, Y 45.0000, Z -3.8333, A 0.000, B 0.000, C 0.000 }
gfCNCPoint3[4292] = {X 121.7693, Y 45.9079, Z -3.8333, A 0.000, B 0.000, C 0.000 }
gfCNCPoint3[4293] = {X 121.4675, Y 46.7702, Z -3.8333, A 0.000, B 0.000, C 0.000 }
gfCNCPoint3[4294] = {X 120.9814, Y 47.5438, Z -3.8333, A 0.000, B 0.000, C 0.000 }
gfCNCPoint3[4295] = {X 120.3354, Y 48.1899, Z -3.8333, A 0.000, B 0.000, C 0.000 }
gfCNCPoint3[4296] = {X 119.5618, Y 48.6760, Z -3.8333, A 0.000, B 0.000, C 0.000 }
gfCNCPoint3[4297] = {X 118.6995, Y 48.9777, Z -3.8333, A 0.000, B 0.000, C 0.000 }
gfCNCPoint3[4298] = {X 117.7916, Y 49.0800, Z -3.8333, A 0.000, B 0.000, C 0.000 }
gfCNCPoint3[4299] = {X 111.9185, Y 49.0800, Z -3.8333, A 0.000, B 0.000, C 0.000 }
gfCNCPoint3[4300] = {X 111.0151, Y 48.9787, Z -3.8333, A 0.000, B 0.000, C 0.000 }
gfCNCPoint3[4301] = {X 110.1565, Y 48.6799, Z -3.8333, A 0.000, B 0.000, C 0.000 }
gfCNCPoint3[4302] = {X 109.3855, Y 48.1985, Z -3.8333, A 0.000, B 0.000, C 0.000 }
gfCNCPoint3[4303] = {X 108.7401, Y 47.5582, Z -3.8333, A 0.000, B 0.000, C 0.000 }
gfCNCPoint3[4304] = {X 108.2526, Y 46.7909, Z -3.8333, A 0.000, B 0.000, C 0.000 }
gfCNCPoint3[4305] = {X 107.9470, Y 45.9348, Z -3.8333, A 0.000, B 0.000, C 0.000 }
gfCNCPoint3[4306] = {X 107.8386, Y 45.0322, Z -3.8333, A 0.000, B 0.000, C 0.000 }
gfCNCPoint3[4307] = {X 107.8385, Y 44.1793, Z -3.8333, A 0.000, B 0.000, C 0.000 }
gfCNCPoint3[4308] = {X 107.8721, Y 43.6672, Z -3.8333, A 0.000, B 0.000, C 0.000 }
gfCNCPoint3[4309] = {X 107.9725, Y 43.1640, Z -3.8333, A 0.000, B 0.000, C 0.000 }
gfCNCPoint3[4310] = {X 108.1299, Y 42.6976, Z -3.8333, A 0.000, B 0.000, C 0.000 }
gfCNCPoint3[4311] = {X 108.3446, Y 42.2547, Z -3.8333, A 0.000, B 0.000, C 0.000 }
gfCNCPoint3[4312] = {X 108.8076, Y 41.5719, Z -3.8333, A 0.000, B 0.000, C 0.000 }
gfCNCPoint3[4313] = {X 109.3663, Y 40.9650, Z -3.8333, A 0.000, B 0.000, C 0.000 }
gfCNCPoint3[4314] = {X 109.3661, Y 39.0029, Z -3.8333, A 0.000, B 0.000, C 0.000 }
gfCNCPoint3[4315] = {X 108.9865, Y 39.0029, Z -3.8333, A 0.000, B 0.000, C 0.000 }
gfCNCPoint3[4316] = {X 105.8902, Y 46.5692, Z -3.8333, A 0.000, B 0.000, C 0.000 }
gfCNCPoint3[4317] = {X 105.5407, Y 47.2300, Z -3.8333, A 0.000, B 0.000, C 0.000 }
gfCNCPoint3[4318] = {X 105.0765, Y 47.8159, Z -3.8333, A 0.000, B 0.000, C 0.000 }
gfCNCPoint3[4319] = {X 104.5133, Y 48.3073, Z -3.8333, A 0.000, B 0.000, C 0.000 }
gfCNCPoint3[4320] = {X 103.8698, Y 48.6877, Z -3.8333, A 0.000, B 0.000, C 0.000 }
gfCNCPoint3[4321] = {X 102.9784, Y 48.9895, Z -3.8333, A 0.000, B 0.000, C 0.000 }
gfCNCPoint3[4322] = {X 102.0417, Y 49.0792, Z -3.8333, A 0.000, B 0.000, C 0.000 }
gfCNCPoint3[4323] = {X 101.1093, Y 48.9518, Z -3.8333, A 0.000, B 0.000, C 0.000 }
gfCNCPoint3[4324] = {X 100.2309, Y 48.6142, Z -3.8333, A 0.000, B 0.000, C 0.000 }
gfCNCPoint3[4325] = {X 99.4532, Y 48.0843, Z -3.8333, A 0.000, B 0.000, C 0.000 }
gfCNCPoint3[4326] = {X 98.8176, Y 47.3903, Z -3.8333, A 0.000, B 0.000, C 0.000 }
gfCNCPoint3[4327] = {X 98.3579, Y 46.5692, Z -3.8333, A 0.000, B 0.000, C 0.000 }
gfCNCPoint3[4328] = {X 94.8918, Y 38.0925, Z -3.8333, A 0.000, B 0.000, C 0.000 }
gfCNCPoint3[4329] = {X 94.8906, Y 38.2310, Z -3.8333, A 0.000, B 0.000, C 0.000 }
gfCNCPoint3[4330] = {X 94.8908, Y 41.0170, Z -3.8333, A 0.000, B 0.000, C 0.000 }
gfCNCPoint3[4331] = {X 95.4387, Y 41.5570, Z -3.8333, A 0.000, B 0.000, C 0.000 }
gfCNCPoint3[4332] = {X 95.8779, Y 42.1885, Z -3.8333, A 0.000, B 0.000, C 0.000 }
gfCNCPoint3[4333] = {X 96.1089, Y 42.6644, Z -3.8333, A 0.000, B 0.000, C 0.000 }
gfCNCPoint3[4334] = {X 96.2776, Y 43.1659, Z -3.8333, A 0.000, B 0.000, C 0.000 }
gfCNCPoint3[4335] = {X 96.3811, Y 43.6826, Z -3.8333, A 0.000, B 0.000, C 0.000 }
gfCNCPoint3[4336] = {X 96.4185, Y 44.2083, Z -3.8333, A 0.000, B 0.000, C 0.000 }
gfCNCPoint3[4337] = {X 96.4184, Y 45.0392, Z -3.8333, A 0.000, B 0.000, C 0.000 }
gfCNCPoint3[4338] = {X 96.3086, Y 45.9406, Z -3.8333, A 0.000, B 0.000, C 0.000 }
gfCNCPoint3[4339] = {X 96.0023, Y 46.7954, Z -3.8333, A 0.000, B 0.000, C 0.000 }
gfCNCPoint3[4340] = {X 95.5144, Y 47.5613, Z -3.8333, A 0.000, B 0.000, C 0.000 }
gfCNCPoint3[4341] = {X 94.8692, Y 48.2003, Z -3.8333, A 0.000, B 0.000, C 0.000 }
gfCNCPoint3[4342] = {X 94.0987, Y 48.6808, Z -3.8333, A 0.000, B 0.000, C 0.000 }
gfCNCPoint3[4343] = {X 93.2410, Y 48.9789, Z -3.8333, A 0.000, B 0.000, C 0.000 }
gfCNCPoint3[4344] = {X 92.3385, Y 49.0800, Z -3.8333, A 0.000, B 0.000, C 0.000 }
gfCNCPoint3[4345] = {X 85.8951, Y 49.0800, Z -3.8333, A 0.000, B 0.000, C 0.000 }
gfCNCPoint3[4346] = {X 84.9918, Y 48.9788, Z -3.8333, A 0.000, B 0.000, C 0.000 }
gfCNCPoint3[4347] = {X 84.1334, Y 48.6801, Z -3.8333, A 0.000, B 0.000, C 0.000 }
gfCNCPoint3[4348] = {X 83.3624, Y 48.1987, Z -3.8333, A 0.000, B 0.000, C 0.000 }
gfCNCPoint3[4349] = {X 82.7171, Y 47.5586, Z -3.8333, A 0.000, B 0.000, C 0.000 }
gfCNCPoint3[4350] = {X 82.2295, Y 46.7916, Z -3.8333, A 0.000, B 0.000, C 0.000 }
gfCNCPoint3[4351] = {X 81.9238, Y 45.9356, Z -3.8333, A 0.000, B 0.000, C 0.000 }
gfCNCPoint3[4352] = {X 81.8152, Y 45.0332, Z -3.8333, A 0.000, B 0.000, C 0.000 }
gfCNCPoint3[4353] = {X 81.8151, Y 44.2084, Z -3.8333, A 0.000, B 0.000, C 0.000 }
gfCNCPoint3[4354] = {X 81.9208, Y 43.3035, Z -3.8333, A 0.000, B 0.000, C 0.000 }
gfCNCPoint3[4355] = {X 82.2219, Y 42.4436, Z -3.8333, A 0.000, B 0.000, C 0.000 }
gfCNCPoint3[4356] = {X 82.7038, Y 41.6705, Z -3.8333, A 0.000, B 0.000, C 0.000 }
gfCNCPoint3[4357] = {X 83.3431, Y 41.0214, Z -3.8333, A 0.000, B 0.000, C 0.000 }
gfCNCPoint3[4358] = {X 83.3430, Y 28.5918, Z -3.8333, A 0.000, B 0.000, C 0.000 }
gfCNCPoint3[4359] = {X 79.3430, Y 28.5918, Z -3.8333, A 0.000, B 0.000, C 0.000 }
gfCNCPoint3[4360] = {X 83.4230, Y 28.5918, Z -3.8333, A 0.000, B 0.000, C 0.000 }
gfCNCPoint3[4361] = {X 83.4228, Y 16.1225, Z -3.8333, A 0.000, B 0.000, C 0.000 }
gfCNCPoint3[4362] = {X 82.7807, Y 15.4882, Z -3.8333, A 0.000, B 0.000, C 0.000 }
gfCNCPoint3[4363] = {X 82.2972, Y 14.7260, Z -3.8333, A 0.000, B 0.000, C 0.000 }
gfCNCPoint3[4364] = {X 81.9969, Y 13.8748, Z -3.8333, A 0.000, B 0.000, C 0.000 }
gfCNCPoint3[4365] = {X 81.8951, Y 12.9779, Z -3.8333, A 0.000, B 0.000, C 0.000 }
gfCNCPoint3[4366] = {X 81.8951, Y 12.1868, Z -3.8333, A 0.000, B 0.000, C 0.000 }
gfCNCPoint3[4367] = {X 81.9954, Y 11.2967, Z -3.8333, A 0.000, B 0.000, C 0.000 }
gfCNCPoint3[4368] = {X 82.2912, Y 10.4513, Z -3.8333, A 0.000, B 0.000, C 0.000 }
gfCNCPoint3[4369] = {X 82.7677, Y 9.6929, Z -3.8333, A 0.000, B 0.000, C 0.000 }
gfCNCPoint3[4370] = {X 83.4011, Y 9.0595, Z -3.8333, A 0.000, B 0.000, C 0.000 }
gfCNCPoint3[4371] = {X 84.1595, Y 8.5829, Z -3.8333, A 0.000, B 0.000, C 0.000 }
gfCNCPoint3[4372] = {X 85.0050, Y 8.2871, Z -3.8333, A 0.000, B 0.000, C 0.000 }
gfCNCPoint3[4373] = {X 85.8951, Y 8.1868, Z -3.8333, A 0.000, B 0.000, C 0.000 }
gfCNCPoint3[4374] = {X 94.0497, Y 8.1868, Z -3.8333, A 0.000, B 0.000, C 0.000 }
gfCNCPoint3[4375] = {X 94.9398, Y 8.2871, Z -3.8333, A 0.000, B 0.000, C 0.000 }
gfCNCPoint3[4376] = {X 95.7852, Y 8.5829, Z -3.8333, A 0.000, B 0.000, C 0.000 }
gfCNCPoint3[4377] = {X 96.5436, Y 9.0595, Z -3.8333, A 0.000, B 0.000, C 0.000 }
gfCNCPoint3[4378] = {X 97.1770, Y 9.6929, Z -3.8333, A 0.000, B 0.000, C 0.000 }
gfCNCPoint3[4379] = {X 97.6535, Y 10.4513, Z -3.8333, A 0.000, B 0.000, C 0.000 }
gfCNCPoint3[4380] = {X 97.9494, Y 11.2967, Z -3.8333, A 0.000, B 0.000, C 0.000 }
gfCNCPoint3[4381] = {X 98.0497, Y 12.1868, Z -3.8333, A 0.000, B 0.000, C 0.000 }
gfCNCPoint3[4382] = {X 98.0495, Y 13.0192, Z -3.8333, A 0.000, B 0.000, C 0.000 }
gfCNCPoint3[4383] = {X 97.9794, Y 13.7246, Z -3.8333, A 0.000, B 0.000, C 0.000 }
gfCNCPoint3[4384] = {X 97.7859, Y 14.4066, Z -3.8333, A 0.000, B 0.000, C 0.000 }
gfCNCPoint3[4385] = {X 97.4750, Y 15.0437, Z -3.8333, A 0.000, B 0.000, C 0.000 }
gfCNCPoint3[4386] = {X 97.4128, Y 15.1435, Z -3.8333, A 0.000, B 0.000, C 0.000 }
gfCNCPoint3[4387] = {X 97.3476, Y 15.2415, Z -3.8333, A 0.000, B 0.000, C 0.000 }
gfCNCPoint3[4388] = {X 97.4108, Y 15.3108, Z -3.8333, A 0.000, B 0.000, C 0.000 }
gfCNCPoint3[4389] = {X 97.9965, Y 16.7687, Z -3.8333, A 0.000, B 0.000, C 0.000 }
gfCNCPoint3[4390] = {X 101.6273, Y 25.7689, Z -3.8333, A 0.000, B 0.000, C 0.000 }
gfCNCPoint3[4391] = {X 101.8768, Y 26.3798, Z -3.8333, A 0.000, B 0.000, C 0.000 }
gfCNCPoint3[4392] = {X 102.1265, Y 25.7689, Z -3.8333, A 0.000, B 0.000, C 0.000 }
gfCNCPoint3[4393] = {X 106.3423, Y 15.2553, Z -3.8333, A 0.000, B 0.000, C 0.000 }
gfCNCPoint3[4394] = {X 106.3813, Y 15.1986, Z -3.8333, A 0.000, B 0.000, C 0.000 }
gfCNCPoint3[4395] = {X 106.3235, Y 15.1096, Z -3.8333, A 0.000, B 0.000, C 0.000 }
gfCNCPoint3[4396] = {X 106.2682, Y 15.0191, Z -3.8333, A 0.000, B 0.000, C 0.000 }
gfCNCPoint3[4397] = {X 105.9605, Y 14.3758, Z -3.8333, A 0.000, B 0.000, C 0.000 }
gfCNCPoint3[4398] = {X 105.7718, Y 13.6882, Z -3.8333, A 0.000, B 0.000, C 0.000 }
gfCNCPoint3[4399] = {X 105.7083, Y 12.9779, Z -3.8333, A 0.000, B 0.000, C 0.000 }
gfCNCPoint3[4400] = {X 105.7083, Y 12.1868, Z -3.8333, A 0.000, B 0.000, C 0.000 }
gfCNCPoint3[4401] = {X 105.8086, Y 11.2967, Z -3.8333, A 0.000, B 0.000, C 0.000 }
gfCNCPoint3[4402] = {X 106.1044, Y 10.4513, Z -3.8333, A 0.000, B 0.000, C 0.000 }
gfCNCPoint3[4403] = {X 106.5810, Y 9.6929, Z -3.8333, A 0.000, B 0.000, C 0.000 }
gfCNCPoint3[4404] = {X 107.2143, Y 9.0595, Z -3.8333, A 0.000, B 0.000, C 0.000 }
gfCNCPoint3[4405] = {X 107.9727, Y 8.5829, Z -3.8333, A 0.000, B 0.000, C 0.000 }
gfCNCPoint3[4406] = {X 108.8182, Y 8.2871, Z -3.8333, A 0.000, B 0.000, C 0.000 }
gfCNCPoint3[4407] = {X 109.7083, Y 8.1868, Z -3.8333, A 0.000, B 0.000, C 0.000 }
gfCNCPoint3[4408] = {X 117.7916, Y 8.1868, Z -3.8333, A 0.000, B 0.000, C 0.000 }
gfCNCPoint3[4409] = {X 118.6817, Y 8.2871, Z -3.8333, A 0.000, B 0.000, C 0.000 }
gfCNCPoint3[4410] = {X 119.5271, Y 8.5829, Z -3.8333, A 0.000, B 0.000, C 0.000 }
gfCNCPoint3[4411] = {X 120.2855, Y 9.0595, Z -3.8333, A 0.000, B 0.000, C 0.000 }
gfCNCPoint3[4412] = {X 120.9189, Y 9.6929, Z -3.8333, A 0.000, B 0.000, C 0.000 }
gfCNCPoint3[4413] = {X 121.3955, Y 10.4513, Z -3.8333, A 0.000, B 0.000, C 0.000 }
gfCNCPoint3[4414] = {X 121.6913, Y 11.2967, Z -3.8333, A 0.000, B 0.000, C 0.000 }
gfCNCPoint3[4415] = {X 121.7916, Y 12.1868, Z -3.8333, A 0.000, B 0.000, C 0.000 }
gfCNCPoint3[4416] = {X 121.7914, Y 13.0192, Z -3.8333, A 0.000, B 0.000, C 0.000 }
gfCNCPoint3[4417] = {X 121.6828, Y 13.9046, Z -3.8333, A 0.000, B 0.000, C 0.000 }
gfCNCPoint3[4418] = {X 121.3807, Y 14.7438, Z -3.8333, A 0.000, B 0.000, C 0.000 }
gfCNCPoint3[4419] = {X 120.9001, Y 15.4953, Z -3.8333, A 0.000, B 0.000, C 0.000 }
gfCNCPoint3[4420] = {X 120.2650, Y 16.1216, Z -3.8333, A 0.000, B 0.000, C 0.000 }
gfCNCPoint3[4421] = {X 120.2637, Y 41.0660, Z -3.8333, A 0.000, B 0.000, C 0.000 }
gfCNCPoint3[4422] = {X 120.4160, Y 41.1901, Z -3.8333, A 0.000, B 0.000, C 0.000 }
gfCNCPoint3[4423] = {X 120.9967, Y 41.8157, Z -3.8333, A 0.000, B 0.000, C 0.000 }
gfCNCPoint3[4424] = {X 121.4315, Y 42.5502, Z -3.8333, A 0.000, B 0.000, C 0.000 }
gfCNCPoint3[4425] = {X 121.7005, Y 43.3602, Z -3.8333, A 0.000, B 0.000, C 0.000 }
gfCNCPoint3[4426] = {X 121.7916, Y 44.2089, Z -3.8333, A 0.000, B 0.000, C 0.000 }
gfCNCPoint3[4427] = {X 121.7916, Y 45.0000, Z -3.8333, A 0.000, B 0.000, C 0.000 }
gfCNCPoint3[4428] = {X 121.6913, Y 45.8901, Z -3.8333, A 0.000, B 0.000, C 0.000 }
gfCNCPoint3[4429] = {X 121.3955, Y 46.7355, Z -3.8333, A 0.000, B 0.000, C 0.000 }
gfCNCPoint3[4430] = {X 120.9189, Y 47.4940, Z -3.8333, A 0.000, B 0.000, C 0.000 }
gfCNCPoint3[4431] = {X 120.2855, Y 48.1273, Z -3.8333, A 0.000, B 0.000, C 0.000 }
gfCNCPoint3[4432] = {X 119.5271, Y 48.6039, Z -3.8333, A 0.000, B 0.000, C 0.000 }
gfCNCPoint3[4433] = {X 118.6817, Y 48.8997, Z -3.8333, A 0.000, B 0.000, C 0.000 }
gfCNCPoint3[4434] = {X 117.7916, Y 49.0000, Z -3.8333, A 0.000, B 0.000, C 0.000 }
gfCNCPoint3[4435] = {X 111.9185, Y 49.0000, Z -3.8333, A 0.000, B 0.000, C 0.000 }
gfCNCPoint3[4436] = {X 111.0284, Y 48.8997, Z -3.8333, A 0.000, B 0.000, C 0.000 }
gfCNCPoint3[4437] = {X 110.1829, Y 48.6039, Z -3.8333, A 0.000, B 0.000, C 0.000 }
gfCNCPoint3[4438] = {X 109.4245, Y 48.1273, Z -3.8333, A 0.000, B 0.000, C 0.000 }
gfCNCPoint3[4439] = {X 108.7911, Y 47.4939, Z -3.8333, A 0.000, B 0.000, C 0.000 }
gfCNCPoint3[4440] = {X 108.3146, Y 46.7355, Z -3.8333, A 0.000, B 0.000, C 0.000 }
gfCNCPoint3[4441] = {X 108.0188, Y 45.8900, Z -3.8333, A 0.000, B 0.000, C 0.000 }
gfCNCPoint3[4442] = {X 107.9185, Y 45.0000, Z -3.8333, A 0.000, B 0.000, C 0.000 }
gfCNCPoint3[4443] = {X 107.9185, Y 44.1793, Z -3.8333, A 0.000, B 0.000, C 0.000 }
gfCNCPoint3[4444] = {X 107.9515, Y 43.6777, Z -3.8333, A 0.000, B 0.000, C 0.000 }
gfCNCPoint3[4445] = {X 108.0498, Y 43.1847, Z -3.8333, A 0.000, B 0.000, C 0.000 }
gfCNCPoint3[4446] = {X 108.2040, Y 42.7279, Z -3.8333, A 0.000, B 0.000, C 0.000 }
gfCNCPoint3[4447] = {X 108.4143, Y 42.2940, Z -3.8333, A 0.000, B 0.000, C 0.000 }
gfCNCPoint3[4448] = {X 108.4389, Y 42.2512, Z -3.8333, A 0.000, B 0.000, C 0.000 }
gfCNCPoint3[4449] = {X 108.4640, Y 42.2086, Z -3.8333, A 0.000, B 0.000, C 0.000 }
gfCNCPoint3[4450] = {X 108.9121, Y 41.5692, Z -3.8333, A 0.000, B 0.000, C 0.000 }
gfCNCPoint3[4451] = {X 109.4463, Y 40.9999, Z -3.8333, A 0.000, B 0.000, C 0.000 }
gfCNCPoint3[4452] = {X 109.4461, Y 38.9229, Z -3.8333, A 0.000, B 0.000, C 0.000 }
gfCNCPoint3[4453] = {X 108.9328, Y 38.9229, Z -3.8333, A 0.000, B 0.000, C 0.000 }
gfCNCPoint3[4454] = {X 105.8164, Y 46.5384, Z -3.8333, A 0.000, B 0.000, C 0.000 }
gfCNCPoint3[4455] = {X 105.3339, Y 47.3869, Z -3.8333, A 0.000, B 0.000, C 0.000 }
gfCNCPoint3[4456] = {X 104.6602, Y 48.0932, Z -3.8333, A 0.000, B 0.000, C 0.000 }
gfCNCPoint3[4457] = {X 103.8355, Y 48.6154, Z -3.8333, A 0.000, B 0.000, C 0.000 }
gfCNCPoint3[4458] = {X 102.9580, Y 48.9121, Z -3.8333, A 0.000, B 0.000, C 0.000 }
gfCNCPoint3[4459] = {X 102.0357, Y 48.9990, Z -3.8333, A 0.000, B 0.000, C 0.000 }
gfCNCPoint3[4460] = {X 101.1182, Y 48.8715, Z -3.8333, A 0.000, B 0.000, C 0.000 }
gfCNCPoint3[4461] = {X 100.2546, Y 48.5362, Z -3.8333, A 0.000, B 0.000, C 0.000 }
gfCNCPoint3[4462] = {X 99.4912, Y 48.0114, Z -3.8333, A 0.000, B 0.000, C 0.000 }
gfCNCPoint3[4463] = {X 98.8691, Y 47.3250, Z -3.8333, A 0.000, B 0.000, C 0.000 }
gfCNCPoint3[4464] = {X 98.4216, Y 46.5139, Z -3.8333, A 0.000, B 0.000, C 0.000 }
gfCNCPoint3[4465] = {X 94.8151, Y 37.6936, Z -3.8333, A 0.000, B 0.000, C 0.000 }
gfCNCPoint3[4466] = {X 94.8106, Y 38.2306, Z -3.8333, A 0.000, B 0.000, C 0.000 }
gfCNCPoint3[4467] = {X 94.8108, Y 41.0552, Z -3.8333, A 0.000, B 0.000, C 0.000 }
gfCNCPoint3[4468] = {X 95.3653, Y 41.5941, Z -3.8333, A 0.000, B 0.000, C 0.000 }
gfCNCPoint3[4469] = {X 95.8083, Y 42.2279, Z -3.8333, A 0.000, B 0.000, C 0.000 }
gfCNCPoint3[4470] = {X 96.0348, Y 42.6947, Z -3.8333, A 0.000, B 0.000, C 0.000 }
gfCNCPoint3[4471] = {X 96.2003, Y 43.1865, Z -3.8333, A 0.000, B 0.000, C 0.000 }
gfCNCPoint3[4472] = {X 96.3018, Y 43.6933, Z -3.8333, A 0.000, B 0.000, C 0.000 }
gfCNCPoint3[4473] = {X 96.3385, Y 44.2089, Z -3.8333, A 0.000, B 0.000, C 0.000 }
gfCNCPoint3[4474] = {X 96.3384, Y 45.0384, Z -3.8333, A 0.000, B 0.000, C 0.000 }
gfCNCPoint3[4475] = {X 96.2308, Y 45.9222, Z -3.8333, A 0.000, B 0.000, C 0.000 }
gfCNCPoint3[4476] = {X 95.9304, Y 46.7602, Z -3.8333, A 0.000, B 0.000, C 0.000 }
gfCNCPoint3[4477] = {X 95.4521, Y 47.5111, Z -3.8333, A 0.000, B 0.000, C 0.000 }
gfCNCPoint3[4478] = {X 94.8196, Y 48.1376, Z -3.8333, A 0.000, B 0.000, C 0.000 }
gfCNCPoint3[4479] = {X 94.0642, Y 48.6086, Z -3.8333, A 0.000, B 0.000, C 0.000 }
gfCNCPoint3[4480] = {X 93.2233, Y 48.9009, Z -3.8333, A 0.000, B 0.000, C 0.000 }
gfCNCPoint3[4481] = {X 92.3385, Y 49.0000, Z -3.8333, A 0.000, B 0.000, C 0.000 }
gfCNCPoint3[4482] = {X 85.8951, Y 49.0000, Z -3.8333, A 0.000, B 0.000, C 0.000 }
gfCNCPoint3[4483] = {X 85.0050, Y 48.8997, Z -3.8333, A 0.000, B 0.000, C 0.000 }
gfCNCPoint3[4484] = {X 84.1595, Y 48.6039, Z -3.8333, A 0.000, B 0.000, C 0.000 }
gfCNCPoint3[4485] = {X 83.4011, Y 48.1273, Z -3.8333, A 0.000, B 0.000, C 0.000 }
gfCNCPoint3[4486] = {X 82.7677, Y 47.4939, Z -3.8333, A 0.000, B 0.000, C 0.000 }
gfCNCPoint3[4487] = {X 82.2912, Y 46.7355, Z -3.8333, A 0.000, B 0.000, C 0.000 }
gfCNCPoint3[4488] = {X 81.9954, Y 45.8901, Z -3.8333, A 0.000, B 0.000, C 0.000 }
gfCNCPoint3[4489] = {X 81.8951, Y 45.0000, Z -3.8333, A 0.000, B 0.000, C 0.000 }
gfCNCPoint3[4490] = {X 81.8951, Y 44.2089, Z -3.8333, A 0.000, B 0.000, C 0.000 }
gfCNCPoint3[4491] = {X 82.0009, Y 43.3122, Z -3.8333, A 0.000, B 0.000, C 0.000 }
gfCNCPoint3[4492] = {X 82.3022, Y 42.4611, Z -3.8333, A 0.000, B 0.000, C 0.000 }
gfCNCPoint3[4493] = {X 82.7843, Y 41.6977, Z -3.8333, A 0.000, B 0.000, C 0.000 }
gfCNCPoint3[4494] = {X 83.4231, Y 41.0597, Z -3.8333, A 0.000, B 0.000, C 0.000 }
gfCNCPoint3[4495] = {X 83.4230, Y 28.5918, Z -3.8333, A 0.000, B 0.000, C 0.000 }
gfCNCPoint3[4496] = {X 79.3430, Y 28.5918, Z -3.8333, A 0.000, B 0.000, C 0.000 }
gfCNCPoint3[4497] = {X 79.3430, Y 28.5918, Z -0.8333, A 0.000, B 0.000, C 0.000 }
gfCNCPoint3[4498] = {X 79.3430, Y 28.5918, Z 11.0000, A 0.000, B 0.000, C 0.000 }
gfCNCPoint3[4499] = {X 136.1636, Y 30.3965, Z 11.0000, A 0.000, B 0.000, C 0.000 }
gfCNCPoint3[4500] = {X 136.1636, Y 30.3965, Z -0.8333, A 0.000, B 0.000, C 0.000 }
gfCNCPoint3[4501] = {X 136.1636, Y 30.3965, Z -3.8333, A 0.000, B 0.000, C 0.000 }
gfCNCPoint3[4502] = {X 140.2436, Y 30.3965, Z -3.8333, A 0.000, B 0.000, C 0.000 }
gfCNCPoint3[4503] = {X 140.2436, Y 19.8772, Z -3.8333, A 0.000, B 0.000, C 0.000 }
gfCNCPoint3[4504] = {X 137.4240, Y 19.8769, Z -3.8333, A 0.000, B 0.000, C 0.000 }
gfCNCPoint3[4505] = {X 136.8916, Y 20.5216, Z -3.8333, A 0.000, B 0.000, C 0.000 }
gfCNCPoint3[4506] = {X 136.2450, Y 21.0517, Z -3.8333, A 0.000, B 0.000, C 0.000 }
gfCNCPoint3[4507] = {X 135.5084, Y 21.4473, Z -3.8333, A 0.000, B 0.000, C 0.000 }
gfCNCPoint3[4508] = {X 134.7093, Y 21.6936, Z -3.8333, A 0.000, B 0.000, C 0.000 }
gfCNCPoint3[4509] = {X 133.8778, Y 21.7814, Z -3.8333, A 0.000, B 0.000, C 0.000 }
gfCNCPoint3[4510] = {X 133.2006, Y 21.7815, Z -3.8333, A 0.000, B 0.000, C 0.000 }
gfCNCPoint3[4511] = {X 132.2394, Y 21.6732, Z -3.8333, A 0.000, B 0.000, C 0.000 }
gfCNCPoint3[4512] = {X 131.3263, Y 21.3537, Z -3.8333, A 0.000, B 0.000, C 0.000 }
gfCNCPoint3[4513] = {X 130.5072, Y 20.8390, Z -3.8333, A 0.000, B 0.000, C 0.000 }
gfCNCPoint3[4514] = {X 129.8231, Y 20.1550, Z -3.8333, A 0.000, B 0.000, C 0.000 }
gfCNCPoint3[4515] = {X 129.3085, Y 19.3359, Z -3.8333, A 0.000, B 0.000, C 0.000 }
gfCNCPoint3[4516] = {X 128.9890, Y 18.4228, Z -3.8333, A 0.000, B 0.000, C 0.000 }
gfCNCPoint3[4517] = {X 128.8806, Y 17.4615, Z -3.8333, A 0.000, B 0.000, C 0.000 }
gfCNCPoint3[4518] = {X 128.8806, Y 10.4835, Z -3.8333, A 0.000, B 0.000, C 0.000 }
gfCNCPoint3[4519] = {X 128.9874, Y 9.5289, Z -3.8333, A 0.000, B 0.000, C 0.000 }
gfCNCPoint3[4520] = {X 129.3026, Y 8.6214, Z -3.8333, A 0.000, B 0.000, C 0.000 }
gfCNCPoint3[4521] = {X 129.8104, Y 7.8061, Z -3.8333, A 0.000, B 0.000, C 0.000 }
gfCNCPoint3[4522] = {X 130.4859, Y 7.1231, Z -3.8333, A 0.000, B 0.000, C 0.000 }
gfCNCPoint3[4523] = {X 131.2956, Y 6.6063, Z -3.8333, A 0.000, B 0.000, C 0.000 }
gfCNCPoint3[4524] = {X 132.1995, Y 6.2811, Z -3.8333, A 0.000, B 0.000, C 0.000 }
gfCNCPoint3[4525] = {X 133.1529, Y 6.1638, Z -3.8333, A 0.000, B 0.000, C 0.000 }
gfCNCPoint3[4526] = {X 133.8866, Y 6.1637, Z -3.8333, A 0.000, B 0.000, C 0.000 }
gfCNCPoint3[4527] = {X 134.7111, Y 6.2518, Z -3.8333, A 0.000, B 0.000, C 0.000 }
gfCNCPoint3[4528] = {X 135.5037, Y 6.4957, Z -3.8333, A 0.000, B 0.000, C 0.000 }
gfCNCPoint3[4529] = {X 136.2350, Y 6.8866, Z -3.8333, A 0.000, B 0.000, C 0.000 }
gfCNCPoint3[4530] = {X 136.8781, Y 7.4100, Z -3.8333, A 0.000, B 0.000, C 0.000 }
gfCNCPoint3[4531] = {X 137.4094, Y 8.0467, Z -3.8333, A 0.000, B 0.000, C 0.000 }
gfCNCPoint3[4532] = {X 155.1125, Y 8.0479, Z -3.8333, A 0.000, B 0.000, C 0.000 }
gfCNCPoint3[4533] = {X 155.6445, Y 7.4101, Z -3.8333, A 0.000, B 0.000, C 0.000 }
gfCNCPoint3[4534] = {X 156.2887, Y 6.8860, Z -3.8333, A 0.000, B 0.000, C 0.000 }
gfCNCPoint3[4535] = {X 157.0214, Y 6.4948, Z -3.8333, A 0.000, B 0.000, C 0.000 }
gfCNCPoint3[4536] = {X 157.8153, Y 6.2510, Z -3.8333, A 0.000, B 0.000, C 0.000 }
gfCNCPoint3[4537] = {X 158.6412, Y 6.1637, Z -3.8333, A 0.000, B 0.000, C 0.000 }
gfCNCPoint3[4538] = {X 159.3781, Y 6.1639, Z -3.8333, A 0.000, B 0.000, C 0.000 }
gfCNCPoint3[4539] = {X 160.3301, Y 6.2828, Z -3.8333, A 0.000, B 0.000, C 0.000 }
gfCNCPoint3[4540] = {X 161.2324, Y 6.6088, Z -3.8333, A 0.000, B 0.000, C 0.000 }
gfCNCPoint3[4541] = {X 162.0405, Y 7.1260, Z -3.8333, A 0.000, B 0.000, C 0.000 }
gfCNCPoint3[4542] = {X 162.7145, Y 7.8088, Z -3.8333, A 0.000, B 0.000, C 0.000 }
gfCNCPoint3[4543] = {X 163.2212, Y 8.6236, Z -3.8333, A 0.000, B 0.000, C 0.000 }
gfCNCPoint3[4544] = {X 163.5355, Y 9.5300, Z -3.8333, A 0.000, B 0.000, C 0.000 }
gfCNCPoint3[4545] = {X 163.6421, Y 10.4835, Z -3.8333, A 0.000, B 0.000, C 0.000 }
gfCNCPoint3[4546] = {X 163.6421, Y 17.4615, Z -3.8333, A 0.000, B 0.000, C 0.000 }
gfCNCPoint3[4547] = {X 163.5355, Y 18.4152, Z -3.8333, A 0.000, B 0.000, C 0.000 }
gfCNCPoint3[4548] = {X 163.2211, Y 19.3218, Z -3.8333, A 0.000, B 0.000, C 0.000 }
gfCNCPoint3[4549] = {X 162.7142, Y 20.1366, Z -3.8333, A 0.000, B 0.000, C 0.000 }
gfCNCPoint3[4550] = {X 162.0400, Y 20.8194, Z -3.8333, A 0.000, B 0.000, C 0.000 }
gfCNCPoint3[4551] = {X 161.2318, Y 21.3365, Z -3.8333, A 0.000, B 0.000, C 0.000 }
gfCNCPoint3[4552] = {X 160.3292, Y 21.6625, Z -3.8333, A 0.000, B 0.000, C 0.000 }
gfCNCPoint3[4553] = {X 159.3770, Y 21.7812, Z -3.8333, A 0.000, B 0.000, C 0.000 }
gfCNCPoint3[4554] = {X 158.6791, Y 21.7815, Z -3.8333, A 0.000, B 0.000, C 0.000 }
gfCNCPoint3[4555] = {X 157.8408, Y 21.6963, Z -3.8333, A 0.000, B 0.000, C 0.000 }
gfCNCPoint3[4556] = {X 157.0346, Y 21.4513, Z -3.8333, A 0.000, B 0.000, C 0.000 }
gfCNCPoint3[4557] = {X 156.2906, Y 21.0556, Z -3.8333, A 0.000, B 0.000, C 0.000 }
gfCNCPoint3[4558] = {X 155.6367, Y 20.5241, Z -3.8333, A 0.000, B 0.000, C 0.000 }
gfCNCPoint3[4559] = {X 155.0974, Y 19.8766, Z -3.8333, A 0.000, B 0.000, C 0.000 }
gfCNCPoint3[4560] = {X 152.2762, Y 19.8779, Z -3.8333, A 0.000, B 0.000, C 0.000 }
gfCNCPoint3[4561] = {X 152.2748, Y 40.8742, Z -3.8333, A 0.000, B 0.000, C 0.000 }
gfCNCPoint3[4562] = {X 152.7409, Y 41.3760, Z -3.8333, A 0.000, B 0.000, C 0.000 }
gfCNCPoint3[4563] = {X 152.8356, Y 41.4889, Z -3.8333, A 0.000, B 0.000, C 0.000 }
gfCNCPoint3[4564] = {X 153.3610, Y 42.3141, Z -3.8333, A 0.000, B 0.000, C 0.000 }
gfCNCPoint3[4565] = {X 153.6890, Y 43.2358, Z -3.8333, A 0.000, B 0.000, C 0.000 }
gfCNCPoint3[4566] = {X 153.8031, Y 44.2075, Z -3.8333, A 0.000, B 0.000, C 0.000 }
gfCNCPoint3[4567] = {X 153.8029, Y 45.0415, Z -3.8333, A 0.000, B 0.000, C 0.000 }
gfCNCPoint3[4568] = {X 153.6867, Y 45.9960, Z -3.8333, A 0.000, B 0.000, C 0.000 }
gfCNCPoint3[4569] = {X 153.3623, Y 46.9011, Z -3.8333, A 0.000, B 0.000, C 0.000 }
gfCNCPoint3[4570] = {X 152.8458, Y 47.7120, Z -3.8333, A 0.000, B 0.000, C 0.000 }
gfCNCPoint3[4571] = {X 152.1626, Y 48.3886, Z -3.8333, A 0.000, B 0.000, C 0.000 }
gfCNCPoint3[4572] = {X 151.3468, Y 48.8973, Z -3.8333, A 0.000, B 0.000, C 0.000 }
gfCNCPoint3[4573] = {X 150.4386, Y 49.2130, Z -3.8333, A 0.000, B 0.000, C 0.000 }
gfCNCPoint3[4574] = {X 149.4831, Y 49.3200, Z -3.8333, A 0.000, B 0.000, C 0.000 }
gfCNCPoint3[4575] = {X 143.0396, Y 49.3200, Z -3.8333, A 0.000, B 0.000, C 0.000 }
gfCNCPoint3[4576] = {X 142.0831, Y 49.2128, Z -3.8333, A 0.000, B 0.000, C 0.000 }
gfCNCPoint3[4577] = {X 141.1741, Y 48.8964, Z -3.8333, A 0.000, B 0.000, C 0.000 }
gfCNCPoint3[4578] = {X 140.3576, Y 48.3866, Z -3.8333, A 0.000, B 0.000, C 0.000 }
gfCNCPoint3[4579] = {X 139.6743, Y 47.7087, Z -3.8333, A 0.000, B 0.000, C 0.000 }
gfCNCPoint3[4580] = {X 139.1581, Y 46.8964, Z -3.8333, A 0.000, B 0.000, C 0.000 }
gfCNCPoint3[4581] = {X 138.8346, Y 45.9899, Z -3.8333, A 0.000, B 0.000, C 0.000 }
gfCNCPoint3[4582] = {X 138.7198, Y 45.0342, Z -3.8333, A 0.000, B 0.000, C 0.000 }
gfCNCPoint3[4583] = {X 138.7200, Y 44.1494, Z -3.8333, A 0.000, B 0.000, C 0.000 }
gfCNCPoint3[4584] = {X 138.8305, Y 43.2364, Z -3.8333, A 0.000, B 0.000, C 0.000 }
gfCNCPoint3[4585] = {X 139.1317, Y 42.3675, Z -3.8333, A 0.000, B 0.000, C 0.000 }
gfCNCPoint3[4586] = {X 139.6099, Y 41.5821, Z -3.8333, A 0.000, B 0.000, C 0.000 }
gfCNCPoint3[4587] = {X 140.2436, Y 40.9157, Z -3.8333, A 0.000, B 0.000, C 0.000 }
gfCNCPoint3[4588] = {X 140.2436, Y 30.3965, Z -3.8333, A 0.000, B 0.000, C 0.000 }
gfCNCPoint3[4589] = {X 136.2436, Y 30.3965, Z -3.8333, A 0.000, B 0.000, C 0.000 }
gfCNCPoint3[4590] = {X 140.3236, Y 30.3965, Z -3.8333, A 0.000, B 0.000, C 0.000 }
gfCNCPoint3[4591] = {X 140.3236, Y 19.7973, Z -3.8333, A 0.000, B 0.000, C 0.000 }
gfCNCPoint3[4592] = {X 137.3798, Y 19.7966, Z -3.8333, A 0.000, B 0.000, C 0.000 }
gfCNCPoint3[4593] = {X 137.3569, Y 19.8333, Z -3.8333, A 0.000, B 0.000, C 0.000 }
gfCNCPoint3[4594] = {X 136.8343, Y 20.4658, Z -3.8333, A 0.000, B 0.000, C 0.000 }
gfCNCPoint3[4595] = {X 136.1998, Y 20.9857, Z -3.8333, A 0.000, B 0.000, C 0.000 }
gfCNCPoint3[4596] = {X 135.4770, Y 21.3738, Z -3.8333, A 0.000, B 0.000, C 0.000 }
gfCNCPoint3[4597] = {X 134.6930, Y 21.6153, Z -3.8333, A 0.000, B 0.000, C 0.000 }
gfCNCPoint3[4598] = {X 133.8772, Y 21.7014, Z -3.8333, A 0.000, B 0.000, C 0.000 }
gfCNCPoint3[4599] = {X 133.2006, Y 21.7015, Z -3.8333, A 0.000, B 0.000, C 0.000 }
gfCNCPoint3[4600] = {X 132.2572, Y 21.5952, Z -3.8333, A 0.000, B 0.000, C 0.000 }
gfCNCPoint3[4601] = {X 131.3610, Y 21.2816, Z -3.8333, A 0.000, B 0.000, C 0.000 }
gfCNCPoint3[4602] = {X 130.5570, Y 20.7765, Z -3.8333, A 0.000, B 0.000, C 0.000 }
gfCNCPoint3[4603] = {X 129.8857, Y 20.1051, Z -3.8333, A 0.000, B 0.000, C 0.000 }
gfCNCPoint3[4604] = {X 129.3805, Y 19.3012, Z -3.8333, A 0.000, B 0.000, C 0.000 }
gfCNCPoint3[4605] = {X 129.0669, Y 18.4050, Z -3.8333, A 0.000, B 0.000, C 0.000 }
gfCNCPoint3[4606] = {X 128.9606, Y 17.4615, Z -3.8333, A 0.000, B 0.000, C 0.000 }
gfCNCPoint3[4607] = {X 128.9606, Y 10.4835, Z -3.8333, A 0.000, B 0.000, C 0.000 }
gfCNCPoint3[4608] = {X 129.0655, Y 9.5466, Z -3.8333, A 0.000, B 0.000, C 0.000 }
gfCNCPoint3[4609] = {X 129.3747, Y 8.6559, Z -3.8333, A 0.000, B 0.000, C 0.000 }
gfCNCPoint3[4610] = {X 129.8732, Y 7.8557, Z -3.8333, A 0.000, B 0.000, C 0.000 }
gfCNCPoint3[4611] = {X 130.5362, Y 7.1853, Z -3.8333, A 0.000, B 0.000, C 0.000 }
gfCNCPoint3[4612] = {X 131.3309, Y 6.6781, Z -3.8333, A 0.000, B 0.000, C 0.000 }
gfCNCPoint3[4613] = {X 132.2180, Y 6.3589, Z -3.8333, A 0.000, B 0.000, C 0.000 }
gfCNCPoint3[4614] = {X 133.1538, Y 6.2438, Z -3.8333, A 0.000, B 0.000, C 0.000 }
gfCNCPoint3[4615] = {X 133.8858, Y 6.2437, Z -3.8333, A 0.000, B 0.000, C 0.000 }
gfCNCPoint3[4616] = {X 134.7033, Y 6.3319, Z -3.8333, A 0.000, B 0.000, C 0.000 }
gfCNCPoint3[4617] = {X 135.4884, Y 6.5761, Z -3.8333, A 0.000, B 0.000, C 0.000 }
gfCNCPoint3[4618] = {X 136.2116, Y 6.9673, Z -3.8333, A 0.000, B 0.000, C 0.000 }
gfCNCPoint3[4619] = {X 136.8458, Y 7.4907, Z -3.8333, A 0.000, B 0.000, C 0.000 }
gfCNCPoint3[4620] = {X 137.3669, Y 8.1267, Z -3.8333, A 0.000, B 0.000, C 0.000 }
gfCNCPoint3[4621] = {X 155.1550, Y 8.1279, Z -3.8333, A 0.000, B 0.000, C 0.000 }
gfCNCPoint3[4622] = {X 155.6769, Y 7.4908, Z -3.8333, A 0.000, B 0.000, C 0.000 }
gfCNCPoint3[4623] = {X 156.3120, Y 6.9667, Z -3.8333, A 0.000, B 0.000, C 0.000 }
gfCNCPoint3[4624] = {X 157.0365, Y 6.5752, Z -3.8333, A 0.000, B 0.000, C 0.000 }
gfCNCPoint3[4625] = {X 157.8231, Y 6.3311, Z -3.8333, A 0.000, B 0.000, C 0.000 }
gfCNCPoint3[4626] = {X 158.6420, Y 6.2437, Z -3.8333, A 0.000, B 0.000, C 0.000 }
gfCNCPoint3[4627] = {X 159.3770, Y 6.2439, Z -3.8333, A 0.000, B 0.000, C 0.000 }
gfCNCPoint3[4628] = {X 160.3114, Y 6.3606, Z -3.8333, A 0.000, B 0.000, C 0.000 }
gfCNCPoint3[4629] = {X 161.1970, Y 6.6806, Z -3.8333, A 0.000, B 0.000, C 0.000 }
gfCNCPoint3[4630] = {X 161.9902, Y 7.1882, Z -3.8333, A 0.000, B 0.000, C 0.000 }
gfCNCPoint3[4631] = {X 162.6517, Y 7.8584, Z -3.8333, A 0.000, B 0.000, C 0.000 }
gfCNCPoint3[4632] = {X 163.1490, Y 8.6580, Z -3.8333, A 0.000, B 0.000, C 0.000 }
gfCNCPoint3[4633] = {X 163.4575, Y 9.5477, Z -3.8333, A 0.000, B 0.000, C 0.000 }
gfCNCPoint3[4634] = {X 163.5621, Y 10.4835, Z -3.8333, A 0.000, B 0.000, C 0.000 }
gfCNCPoint3[4635] = {X 163.5621, Y 17.4615, Z -3.8333, A 0.000, B 0.000, C 0.000 }
gfCNCPoint3[4636] = {X 163.4575, Y 18.3975, Z -3.8333, A 0.000, B 0.000, C 0.000 }
gfCNCPoint3[4637] = {X 163.1489, Y 19.2873, Z -3.8333, A 0.000, B 0.000, C 0.000 }
gfCNCPoint3[4638] = {X 162.6514, Y 20.0870, Z -3.8333, A 0.000, B 0.000, C 0.000 }
gfCNCPoint3[4639] = {X 161.9897, Y 20.7572, Z -3.8333, A 0.000, B 0.000, C 0.000 }
gfCNCPoint3[4640] = {X 161.1964, Y 21.2648, Z -3.8333, A 0.000, B 0.000, C 0.000 }
gfCNCPoint3[4641] = {X 160.3106, Y 21.5847, Z -3.8333, A 0.000, B 0.000, C 0.000 }
gfCNCPoint3[4642] = {X 159.3760, Y 21.7012, Z -3.8333, A 0.000, B 0.000, C 0.000 }
gfCNCPoint3[4643] = {X 158.6795, Y 21.7015, Z -3.8333, A 0.000, B 0.000, C 0.000 }
gfCNCPoint3[4644] = {X 157.8483, Y 21.6162, Z -3.8333, A 0.000, B 0.000, C 0.000 }
gfCNCPoint3[4645] = {X 157.0495, Y 21.3709, Z -3.8333, A 0.000, B 0.000, C 0.000 }
gfCNCPoint3[4646] = {X 156.3138, Y 20.9749, Z -3.8333, A 0.000, B 0.000, C 0.000 }
gfCNCPoint3[4647] = {X 155.6690, Y 20.4434, Z -3.8333, A 0.000, B 0.000, C 0.000 }
gfCNCPoint3[4648] = {X 155.1400, Y 19.7966, Z -3.8333, A 0.000, B 0.000, C 0.000 }
gfCNCPoint3[4649] = {X 152.1962, Y 19.7979, Z -3.8333, A 0.000, B 0.000, C 0.000 }
gfCNCPoint3[4650] = {X 152.1948, Y 40.9056, Z -3.8333, A 0.000, B 0.000, C 0.000 }
gfCNCPoint3[4651] = {X 152.6809, Y 41.4289, Z -3.8333, A 0.000, B 0.000, C 0.000 }
gfCNCPoint3[4652] = {X 152.7738, Y 41.5397, Z -3.8333, A 0.000, B 0.000, C 0.000 }
gfCNCPoint3[4653] = {X 153.2893, Y 42.3497, Z -3.8333, A 0.000, B 0.000, C 0.000 }
gfCNCPoint3[4654] = {X 153.6112, Y 43.2543, Z -3.8333, A 0.000, B 0.000, C 0.000 }
gfCNCPoint3[4655] = {X 153.7231, Y 44.2079, Z -3.8333, A 0.000, B 0.000, C 0.000 }
gfCNCPoint3[4656] = {X 153.7229, Y 45.0408, Z -3.8333, A 0.000, B 0.000, C 0.000 }
gfCNCPoint3[4657] = {X 153.6089, Y 45.9775, Z -3.8333, A 0.000, B 0.000, C 0.000 }
gfCNCPoint3[4658] = {X 153.2905, Y 46.8659, Z -3.8333, A 0.000, B 0.000, C 0.000 }
gfCNCPoint3[4659] = {X 152.7835, Y 47.6618, Z -3.8333, A 0.000, B 0.000, C 0.000 }
gfCNCPoint3[4660] = {X 152.1130, Y 48.3258, Z -3.8333, A 0.000, B 0.000, C 0.000 }
gfCNCPoint3[4661] = {X 151.3123, Y 48.8251, Z -3.8333, A 0.000, B 0.000, C 0.000 }
gfCNCPoint3[4662] = {X 150.4209, Y 49.1350, Z -3.8333, A 0.000, B 0.000, C 0.000 }
gfCNCPoint3[4663] = {X 149.4831, Y 49.2400, Z -3.8333, A 0.000, B 0.000, C 0.000 }
gfCNCPoint3[4664] = {X 143.0396, Y 49.2400, Z -3.8333, A 0.000, B 0.000, C 0.000 }
gfCNCPoint3[4665] = {X 142.1008, Y 49.1348, Z -3.8333, A 0.000, B 0.000, C 0.000 }
gfCNCPoint3[4666] = {X 141.2086, Y 48.8243, Z -3.8333, A 0.000, B 0.000, C 0.000 }
gfCNCPoint3[4667] = {X 140.4073, Y 48.3239, Z -3.8333, A 0.000, B 0.000, C 0.000 }
gfCNCPoint3[4668] = {X 139.7367, Y 47.6586, Z -3.8333, A 0.000, B 0.000, C 0.000 }
gfCNCPoint3[4669] = {X 139.2300, Y 46.8612, Z -3.8333, A 0.000, B 0.000, C 0.000 }
gfCNCPoint3[4670] = {X 138.9124, Y 45.9715, Z -3.8333, A 0.000, B 0.000, C 0.000 }
gfCNCPoint3[4671] = {X 138.7998, Y 45.0336, Z -3.8333, A 0.000, B 0.000, C 0.000 }
gfCNCPoint3[4672] = {X 138.8000, Y 44.1505, Z -3.8333, A 0.000, B 0.000, C 0.000 }
gfCNCPoint3[4673] = {X 138.9105, Y 43.2454, Z -3.8333, A 0.000, B 0.000, C 0.000 }
gfCNCPoint3[4674] = {X 139.2119, Y 42.3850, Z -3.8333, A 0.000, B 0.000, C 0.000 }
gfCNCPoint3[4675] = {X 139.6903, Y 41.6088, Z -3.8333, A 0.000, B 0.000, C 0.000 }
gfCNCPoint3[4676] = {X 140.3236, Y 40.9529, Z -3.8333, A 0.000, B 0.000, C 0.000 }
gfCNCPoint3[4677] = {X 140.3236, Y 30.3965, Z -3.8333, A 0.000, B 0.000, C 0.000 }
gfCNCPoint3[4678] = {X 136.3236, Y 30.3965, Z -3.8333, A 0.000, B 0.000, C 0.000 }
gfCNCPoint3[4679] = {X 140.4036, Y 30.3965, Z -3.8333, A 0.000, B 0.000, C 0.000 }
gfCNCPoint3[4680] = {X 140.4036, Y 19.7173, Z -3.8333, A 0.000, B 0.000, C 0.000 }
gfCNCPoint3[4681] = {X 137.3353, Y 19.7165, Z -3.8333, A 0.000, B 0.000, C 0.000 }
gfCNCPoint3[4682] = {X 137.2897, Y 19.7898, Z -3.8333, A 0.000, B 0.000, C 0.000 }
gfCNCPoint3[4683] = {X 136.7771, Y 20.4099, Z -3.8333, A 0.000, B 0.000, C 0.000 }
gfCNCPoint3[4684] = {X 136.1546, Y 20.9197, Z -3.8333, A 0.000, B 0.000, C 0.000 }
gfCNCPoint3[4685] = {X 135.4456, Y 21.3002, Z -3.8333, A 0.000, B 0.000, C 0.000 }
gfCNCPoint3[4686] = {X 134.6767, Y 21.5370, Z -3.8333, A 0.000, B 0.000, C 0.000 }
gfCNCPoint3[4687] = {X 133.8765, Y 21.6214, Z -3.8333, A 0.000, B 0.000, C 0.000 }
gfCNCPoint3[4688] = {X 133.2006, Y 21.6215, Z -3.8333, A 0.000, B 0.000, C 0.000 }
gfCNCPoint3[4689] = {X 132.2750, Y 21.5172, Z -3.8333, A 0.000, B 0.000, C 0.000 }
gfCNCPoint3[4690] = {X 131.3957, Y 21.2096, Z -3.8333, A 0.000, B 0.000, C 0.000 }
gfCNCPoint3[4691] = {X 130.6069, Y 20.7140, Z -3.8333, A 0.000, B 0.000, C 0.000 }
gfCNCPoint3[4692] = {X 129.9482, Y 20.0553, Z -3.8333, A 0.000, B 0.000, C 0.000 }
gfCNCPoint3[4693] = {X 129.4526, Y 19.2665, Z -3.8333, A 0.000, B 0.000, C 0.000 }
gfCNCPoint3[4694] = {X 129.1449, Y 18.3872, Z -3.8333, A 0.000, B 0.000, C 0.000 }
gfCNCPoint3[4695] = {X 129.0406, Y 17.4615, Z -3.8333, A 0.000, B 0.000, C 0.000 }
gfCNCPoint3[4696] = {X 129.0406, Y 10.4835, Z -3.8333, A 0.000, B 0.000, C 0.000 }
gfCNCPoint3[4697] = {X 129.1435, Y 9.5642, Z -3.8333, A 0.000, B 0.000, C 0.000 }
gfCNCPoint3[4698] = {X 129.4469, Y 8.6904, Z -3.8333, A 0.000, B 0.000, C 0.000 }
gfCNCPoint3[4699] = {X 129.9360, Y 7.9052, Z -3.8333, A 0.000, B 0.000, C 0.000 }
gfCNCPoint3[4700] = {X 130.5864, Y 7.2475, Z -3.8333, A 0.000, B 0.000, C 0.000 }
gfCNCPoint3[4701] = {X 131.3662, Y 6.7499, Z -3.8333, A 0.000, B 0.000, C 0.000 }
gfCNCPoint3[4702] = {X 132.2366, Y 6.4368, Z -3.8333, A 0.000, B 0.000, C 0.000 }
gfCNCPoint3[4703] = {X 133.1547, Y 6.3238, Z -3.8333, A 0.000, B 0.000, C 0.000 }
gfCNCPoint3[4704] = {X 133.8850, Y 6.3237, Z -3.8333, A 0.000, B 0.000, C 0.000 }
gfCNCPoint3[4705] = {X 134.6954, Y 6.4119, Z -3.8333, A 0.000, B 0.000, C 0.000 }
gfCNCPoint3[4706] = {X 135.4730, Y 6.6565, Z -3.8333, A 0.000, B 0.000, C 0.000 }
gfCNCPoint3[4707] = {X 136.1881, Y 7.0480, Z -3.8333, A 0.000, B 0.000, C 0.000 }
gfCNCPoint3[4708] = {X 136.8131, Y 7.5714, Z -3.8333, A 0.000, B 0.000, C 0.000 }
gfCNCPoint3[4709] = {X 137.3239, Y 8.2067, Z -3.8333, A 0.000, B 0.000, C 0.000 }
gfCNCPoint3[4710] = {X 155.1980, Y 8.2079, Z -3.8333, A 0.000, B 0.000, C 0.000 }
gfCNCPoint3[4711] = {X 155.7096, Y 7.5715, Z -3.8333, A 0.000, B 0.000, C 0.000 }
gfCNCPoint3[4712] = {X 156.3355, Y 7.0474, Z -3.8333, A 0.000, B 0.000, C 0.000 }
gfCNCPoint3[4713] = {X 157.0519, Y 6.6555, Z -3.8333, A 0.000, B 0.000, C 0.000 }
gfCNCPoint3[4714] = {X 157.8309, Y 6.4112, Z -3.8333, A 0.000, B 0.000, C 0.000 }
gfCNCPoint3[4715] = {X 158.6427, Y 6.3237, Z -3.8333, A 0.000, B 0.000, C 0.000 }
gfCNCPoint3[4716] = {X 159.3760, Y 6.3239, Z -3.8333, A 0.000, B 0.000, C 0.000 }
gfCNCPoint3[4717] = {X 160.2928, Y 6.4383, Z -3.8333, A 0.000, B 0.000, C 0.000 }
gfCNCPoint3[4718] = {X 161.1617, Y 6.7524, Z -3.8333, A 0.000, B 0.000, C 0.000 }
gfCNCPoint3[4719] = {X 161.9398, Y 7.2504, Z -3.8333, A 0.000, B 0.000, C 0.000 }
gfCNCPoint3[4720] = {X 162.5889, Y 7.9079, Z -3.8333, A 0.000, B 0.000, C 0.000 }
gfCNCPoint3[4721] = {X 163.0768, Y 8.6925, Z -3.8333, A 0.000, B 0.000, C 0.000 }
gfCNCPoint3[4722] = {X 163.3795, Y 9.5653, Z -3.8333, A 0.000, B 0.000, C 0.000 }
gfCNCPoint3[4723] = {X 163.4821, Y 10.4835, Z -3.8333, A 0.000, B 0.000, C 0.000 }
gfCNCPoint3[4724] = {X 163.4821, Y 17.4615, Z -3.8333, A 0.000, B 0.000, C 0.000 }
gfCNCPoint3[4725] = {X 163.3795, Y 18.3798, Z -3.8333, A 0.000, B 0.000, C 0.000 }
gfCNCPoint3[4726] = {X 163.0767, Y 19.2527, Z -3.8333, A 0.000, B 0.000, C 0.000 }
gfCNCPoint3[4727] = {X 162.5887, Y 20.0373, Z -3.8333, A 0.000, B 0.000, C 0.000 }
gfCNCPoint3[4728] = {X 161.9396, Y 20.6948, Z -3.8333, A 0.000, B 0.000, C 0.000 }
gfCNCPoint3[4729] = {X 161.1613, Y 21.1929, Z -3.8333, A 0.000, B 0.000, C 0.000 }
gfCNCPoint3[4730] = {X 160.2923, Y 21.5068, Z -3.8333, A 0.000, B 0.000, C 0.000 }
gfCNCPoint3[4731] = {X 159.3755, Y 21.6212, Z -3.8333, A 0.000, B 0.000, C 0.000 }
gfCNCPoint3[4732] = {X 158.6798, Y 21.6215, Z -3.8333, A 0.000, B 0.000, C 0.000 }
gfCNCPoint3[4733] = {X 157.8558, Y 21.5361, Z -3.8333, A 0.000, B 0.000, C 0.000 }
gfCNCPoint3[4734] = {X 157.0646, Y 21.2904, Z -3.8333, A 0.000, B 0.000, C 0.000 }
gfCNCPoint3[4735] = {X 156.3371, Y 20.8941, Z -3.8333, A 0.000, B 0.000, C 0.000 }
gfCNCPoint3[4736] = {X 155.7017, Y 20.3626, Z -3.8333, A 0.000, B 0.000, C 0.000 }
gfCNCPoint3[4737] = {X 155.1831, Y 19.7166, Z -3.8333, A 0.000, B 0.000, C 0.000 }
gfCNCPoint3[4738] = {X 152.1162, Y 19.7179, Z -3.8333, A 0.000, B 0.000, C 0.000 }
gfCNCPoint3[4739] = {X 152.1148, Y 40.9370, Z -3.8333, A 0.000, B 0.000, C 0.000 }
gfCNCPoint3[4740] = {X 152.6209, Y 41.4819, Z -3.8333, A 0.000, B 0.000, C 0.000 }
gfCNCPoint3[4741] = {X 152.7120, Y 41.5905, Z -3.8333, A 0.000, B 0.000, C 0.000 }
gfCNCPoint3[4742] = {X 153.2177, Y 42.3852, Z -3.8333, A 0.000, B 0.000, C 0.000 }
gfCNCPoint3[4743] = {X 153.5333, Y 43.2727, Z -3.8333, A 0.000, B 0.000, C 0.000 }
gfCNCPoint3[4744] = {X 153.6431, Y 44.2082, Z -3.8333, A 0.000, B 0.000, C 0.000 }
gfCNCPoint3[4745] = {X 153.6429, Y 45.0400, Z -3.8333, A 0.000, B 0.000, C 0.000 }
gfCNCPoint3[4746] = {X 153.5310, Y 45.9591, Z -3.8333, A 0.000, B 0.000, C 0.000 }
gfCNCPoint3[4747] = {X 153.2186, Y 46.8306, Z -3.8333, A 0.000, B 0.000, C 0.000 }
gfCNCPoint3[4748] = {X 152.7212, Y 47.6115, Z -3.8333, A 0.000, B 0.000, C 0.000 }
gfCNCPoint3[4749] = {X 152.0634, Y 48.2631, Z -3.8333, A 0.000, B 0.000, C 0.000 }
gfCNCPoint3[4750] = {X 151.2778, Y 48.7530, Z -3.8333, A 0.000, B 0.000, C 0.000 }
gfCNCPoint3[4751] = {X 150.4032, Y 49.0570, Z -3.8333, A 0.000, B 0.000, C 0.000 }
gfCNCPoint3[4752] = {X 149.4831, Y 49.1600, Z -3.8333, A 0.000, B 0.000, C 0.000 }
gfCNCPoint3[4753] = {X 143.0396, Y 49.1600, Z -3.8333, A 0.000, B 0.000, C 0.000 }
gfCNCPoint3[4754] = {X 142.1185, Y 49.0567, Z -3.8333, A 0.000, B 0.000, C 0.000 }
gfCNCPoint3[4755] = {X 141.2432, Y 48.7521, Z -3.8333, A 0.000, B 0.000, C 0.000 }
gfCNCPoint3[4756] = {X 140.4570, Y 48.2612, Z -3.8333, A 0.000, B 0.000, C 0.000 }
gfCNCPoint3[4757] = {X 139.7990, Y 47.6084, Z -3.8333, A 0.000, B 0.000, C 0.000 }
gfCNCPoint3[4758] = {X 139.3019, Y 46.8261, Z -3.8333, A 0.000, B 0.000, C 0.000 }
gfCNCPoint3[4759] = {X 138.9903, Y 45.9532, Z -3.8333, A 0.000, B 0.000, C 0.000 }
gfCNCPoint3[4760] = {X 138.8798, Y 45.0329, Z -3.8333, A 0.000, B 0.000, C 0.000 }
gfCNCPoint3[4761] = {X 138.8800, Y 44.1516, Z -3.8333, A 0.000, B 0.000, C 0.000 }
gfCNCPoint3[4762] = {X 138.9906, Y 43.2545, Z -3.8333, A 0.000, B 0.000, C 0.000 }
gfCNCPoint3[4763] = {X 139.2922, Y 42.4026, Z -3.8333, A 0.000, B 0.000, C 0.000 }
gfCNCPoint3[4764] = {X 139.7708, Y 41.6358, Z -3.8333, A 0.000, B 0.000, C 0.000 }
gfCNCPoint3[4765] = {X 140.4036, Y 40.9906, Z -3.8333, A 0.000, B 0.000, C 0.000 }
gfCNCPoint3[4766] = {X 140.4036, Y 30.3965, Z -3.8333, A 0.000, B 0.000, C 0.000 }
gfCNCPoint3[4767] = {X 136.4036, Y 30.3965, Z -3.8333, A 0.000, B 0.000, C 0.000 }
gfCNCPoint3[4768] = {X 140.4836, Y 30.3965, Z -3.8333, A 0.000, B 0.000, C 0.000 }
gfCNCPoint3[4769] = {X 140.4836, Y 19.6373, Z -3.8333, A 0.000, B 0.000, C 0.000 }
gfCNCPoint3[4770] = {X 137.2909, Y 19.6365, Z -3.8333, A 0.000, B 0.000, C 0.000 }
gfCNCPoint3[4771] = {X 137.2218, Y 19.7475, Z -3.8333, A 0.000, B 0.000, C 0.000 }
gfCNCPoint3[4772] = {X 136.5756, Y 20.4907, Z -3.8333, A 0.000, B 0.000, C 0.000 }
gfCNCPoint3[4773] = {X 135.7702, Y 21.0573, Z -3.8333, A 0.000, B 0.000, C 0.000 }
gfCNCPoint3[4774] = {X 134.8524, Y 21.4145, Z -3.8333, A 0.000, B 0.000, C 0.000 }
gfCNCPoint3[4775] = {X 133.8758, Y 21.5414, Z -3.8333, A 0.000, B 0.000, C 0.000 }
gfCNCPoint3[4776] = {X 133.2006, Y 21.5415, Z -3.8333, A 0.000, B 0.000, C 0.000 }
gfCNCPoint3[4777] = {X 132.2928, Y 21.4392, Z -3.8333, A 0.000, B 0.000, C 0.000 }
gfCNCPoint3[4778] = {X 131.4304, Y 21.1375, Z -3.8333, A 0.000, B 0.000, C 0.000 }
gfCNCPoint3[4779] = {X 130.6568, Y 20.6514, Z -3.8333, A 0.000, B 0.000, C 0.000 }
gfCNCPoint3[4780] = {X 130.0108, Y 20.0054, Z -3.8333, A 0.000, B 0.000, C 0.000 }
gfCNCPoint3[4781] = {X 129.5247, Y 19.2318, Z -3.8333, A 0.000, B 0.000, C 0.000 }
gfCNCPoint3[4782] = {X 129.2229, Y 18.3694, Z -3.8333, A 0.000, B 0.000, C 0.000 }
gfCNCPoint3[4783] = {X 129.1206, Y 17.4615, Z -3.8333, A 0.000, B 0.000, C 0.000 }
gfCNCPoint3[4784] = {X 129.1206, Y 10.4835, Z -3.8333, A 0.000, B 0.000, C 0.000 }
gfCNCPoint3[4785] = {X 129.2215, Y 9.5820, Z -3.8333, A 0.000, B 0.000, C 0.000 }
gfCNCPoint3[4786] = {X 129.5191, Y 8.7250, Z -3.8333, A 0.000, B 0.000, C 0.000 }
gfCNCPoint3[4787] = {X 129.9986, Y 7.9550, Z -3.8333, A 0.000, B 0.000, C 0.000 }
gfCNCPoint3[4788] = {X 130.6365, Y 7.3099, Z -3.8333, A 0.000, B 0.000, C 0.000 }
gfCNCPoint3[4789] = {X 131.4011, Y 6.8218, Z -3.8333, A 0.000, B 0.000, C 0.000 }
gfCNCPoint3[4790] = {X 132.2547, Y 6.5147, Z -3.8333, A 0.000, B 0.000, C 0.000 }
gfCNCPoint3[4791] = {X 133.1551, Y 6.4038, Z -3.8333, A 0.000, B 0.000, C 0.000 }
gfCNCPoint3[4792] = {X 133.8841, Y 6.4037, Z -3.8333, A 0.000, B 0.000, C 0.000 }
gfCNCPoint3[4793] = {X 134.6874, Y 6.4920, Z -3.8333, A 0.000, B 0.000, C 0.000 }
gfCNCPoint3[4794] = {X 135.4575, Y 6.7369, Z -3.8333, A 0.000, B 0.000, C 0.000 }
gfCNCPoint3[4795] = {X 136.1643, Y 7.1287, Z -3.8333, A 0.000, B 0.000, C 0.000 }
gfCNCPoint3[4796] = {X 136.7800, Y 7.6522, Z -3.8333, A 0.000, B 0.000, C 0.000 }
gfCNCPoint3[4797] = {X 137.2804, Y 8.2867, Z -3.8333, A 0.000, B 0.000, C 0.000 }
gfCNCPoint3[4798] = {X 155.2416, Y 8.2879, Z -3.8333, A 0.000, B 0.000, C 0.000 }
gfCNCPoint3[4799] = {X 155.2870, Y 8.2183, Z -3.8333, A 0.000, B 0.000, C 0.000 }
gfCNCPoint3[4800] = {X 155.3338, Y 8.1497, Z -3.8333, A 0.000, B 0.000, C 0.000 }
gfCNCPoint3[4801] = {X 155.9789, Y 7.4260, Z -3.8333, A 0.000, B 0.000, C 0.000 }
gfCNCPoint3[4802] = {X 156.7766, Y 6.8749, Z -3.8333, A 0.000, B 0.000, C 0.000 }
gfCNCPoint3[4803] = {X 157.6818, Y 6.5276, Z -3.8333, A 0.000, B 0.000, C 0.000 }
gfCNCPoint3[4804] = {X 158.6434, Y 6.4037, Z -3.8333, A 0.000, B 0.000, C 0.000 }
gfCNCPoint3[4805] = {X 159.3750, Y 6.4039, Z -3.8333, A 0.000, B 0.000, C 0.000 }
gfCNCPoint3[4806] = {X 160.2741, Y 6.5161, Z -3.8333, A 0.000, B 0.000, C 0.000 }
gfCNCPoint3[4807] = {X 161.1263, Y 6.8241, Z -3.8333, A 0.000, B 0.000, C 0.000 }
gfCNCPoint3[4808] = {X 161.8895, Y 7.3126, Z -3.8333, A 0.000, B 0.000, C 0.000 }
gfCNCPoint3[4809] = {X 162.5260, Y 7.9574, Z -3.8333, A 0.000, B 0.000, C 0.000 }
gfCNCPoint3[4810] = {X 163.0046, Y 8.7269, Z -3.8333, A 0.000, B 0.000, C 0.000 }
gfCNCPoint3[4811] = {X 163.3015, Y 9.5830, Z -3.8333, A 0.000, B 0.000, C 0.000 }
gfCNCPoint3[4812] = {X 163.4021, Y 10.4835, Z -3.8333, A 0.000, B 0.000, C 0.000 }
gfCNCPoint3[4813] = {X 163.4021, Y 17.4615, Z -3.8333, A 0.000, B 0.000, C 0.000 }
gfCNCPoint3[4814] = {X 163.3015, Y 18.3621, Z -3.8333, A 0.000, B 0.000, C 0.000 }
gfCNCPoint3[4815] = {X 163.0046, Y 19.2182, Z -3.8333, A 0.000, B 0.000, C 0.000 }
gfCNCPoint3[4816] = {X 162.5260, Y 19.9876, Z -3.8333, A 0.000, B 0.000, C 0.000 }
gfCNCPoint3[4817] = {X 161.8895, Y 20.6325, Z -3.8333, A 0.000, B 0.000, C 0.000 }
gfCNCPoint3[4818] = {X 161.1263, Y 21.1209, Z -3.8333, A 0.000, B 0.000, C 0.000 }
gfCNCPoint3[4819] = {X 160.2741, Y 21.4289, Z -3.8333, A 0.000, B 0.000, C 0.000 }
gfCNCPoint3[4820] = {X 159.3750, Y 21.5412, Z -3.8333, A 0.000, B 0.000, C 0.000 }
gfCNCPoint3[4821] = {X 158.6802, Y 21.5415, Z -3.8333, A 0.000, B 0.000, C 0.000 }
gfCNCPoint3[4822] = {X 157.8634, Y 21.4560, Z -3.8333, A 0.000, B 0.000, C 0.000 }
gfCNCPoint3[4823] = {X 157.0799, Y 21.2100, Z -3.8333, A 0.000, B 0.000, C 0.000 }
gfCNCPoint3[4824] = {X 156.3608, Y 20.8133, Z -3.8333, A 0.000, B 0.000, C 0.000 }
gfCNCPoint3[4825] = {X 155.7347, Y 20.2818, Z -3.8333, A 0.000, B 0.000, C 0.000 }
gfCNCPoint3[4826] = {X 155.2267, Y 19.6366, Z -3.8333, A 0.000, B 0.000, C 0.000 }
gfCNCPoint3[4827] = {X 152.0362, Y 19.6380, Z -3.8333, A 0.000, B 0.000, C 0.000 }
gfCNCPoint3[4828] = {X 152.0348, Y 40.9684, Z -3.8333, A 0.000, B 0.000, C 0.000 }
gfCNCPoint3[4829] = {X 152.5609, Y 41.5348, Z -3.8333, A 0.000, B 0.000, C 0.000 }
gfCNCPoint3[4830] = {X 152.6502, Y 41.6414, Z -3.8333, A 0.000, B 0.000, C 0.000 }
gfCNCPoint3[4831] = {X 153.1460, Y 42.4208, Z -3.8333, A 0.000, B 0.000, C 0.000 }
gfCNCPoint3[4832] = {X 153.4555, Y 43.2911, Z -3.8333, A 0.000, B 0.000, C 0.000 }
gfCNCPoint3[4833] = {X 153.5631, Y 44.2085, Z -3.8333, A 0.000, B 0.000, C 0.000 }
gfCNCPoint3[4834] = {X 153.5629, Y 45.0392, Z -3.8333, A 0.000, B 0.000, C 0.000 }
gfCNCPoint3[4835] = {X 153.4532, Y 45.9406, Z -3.8333, A 0.000, B 0.000, C 0.000 }
gfCNCPoint3[4836] = {X 153.1468, Y 46.7954, Z -3.8333, A 0.000, B 0.000, C 0.000 }
gfCNCPoint3[4837] = {X 152.6589, Y 47.5613, Z -3.8333, A 0.000, B 0.000, C 0.000 }
gfCNCPoint3[4838] = {X 152.0138, Y 48.2003, Z -3.8333, A 0.000, B 0.000, C 0.000 }
gfCNCPoint3[4839] = {X 151.2432, Y 48.6808, Z -3.8333, A 0.000, B 0.000, C 0.000 }
gfCNCPoint3[4840] = {X 150.3855, Y 48.9789, Z -3.8333, A 0.000, B 0.000, C 0.000 }
gfCNCPoint3[4841] = {X 149.4831, Y 49.0800, Z -3.8333, A 0.000, B 0.000, C 0.000 }
gfCNCPoint3[4842] = {X 143.0396, Y 49.0800, Z -3.8333, A 0.000, B 0.000, C 0.000 }
gfCNCPoint3[4843] = {X 142.1362, Y 48.9787, Z -3.8333, A 0.000, B 0.000, C 0.000 }
gfCNCPoint3[4844] = {X 141.2777, Y 48.6799, Z -3.8333, A 0.000, B 0.000, C 0.000 }
gfCNCPoint3[4845] = {X 140.5066, Y 48.1985, Z -3.8333, A 0.000, B 0.000, C 0.000 }
gfCNCPoint3[4846] = {X 139.8613, Y 47.5582, Z -3.8333, A 0.000, B 0.000, C 0.000 }
gfCNCPoint3[4847] = {X 139.3737, Y 46.7910, Z -3.8333, A 0.000, B 0.000, C 0.000 }
gfCNCPoint3[4848] = {X 139.0682, Y 45.9349, Z -3.8333, A 0.000, B 0.000, C 0.000 }
gfCNCPoint3[4849] = {X 138.9598, Y 45.0323, Z -3.8333, A 0.000, B 0.000, C 0.000 }
gfCNCPoint3[4850] = {X 138.9600, Y 44.1527, Z -3.8333, A 0.000, B 0.000, C 0.000 }
gfCNCPoint3[4851] = {X 139.0706, Y 43.2637, Z -3.8333, A 0.000, B 0.000, C 0.000 }
gfCNCPoint3[4852] = {X 139.3725, Y 42.4203, Z -3.8333, A 0.000, B 0.000, C 0.000 }
gfCNCPoint3[4853] = {X 139.8512, Y 41.6631, Z -3.8333, A 0.000, B 0.000, C 0.000 }
gfCNCPoint3[4854] = {X 140.4836, Y 41.0287, Z -3.8333, A 0.000, B 0.000, C 0.000 }
gfCNCPoint3[4855] = {X 140.4836, Y 30.3965, Z -3.8333, A 0.000, B 0.000, C 0.000 }
gfCNCPoint3[4856] = {X 136.4836, Y 30.3965, Z -3.8333, A 0.000, B 0.000, C 0.000 }
gfCNCPoint3[4857] = {X 140.5636, Y 30.3965, Z -3.8333, A 0.000, B 0.000, C 0.000 }
gfCNCPoint3[4858] = {X 140.5636, Y 19.9572, Z -3.8333, A 0.000, B 0.000, C 0.000 }
gfCNCPoint3[4859] = {X 140.5645, Y 19.5573, Z -3.8333, A 0.000, B 0.000, C 0.000 }
gfCNCPoint3[4860] = {X 137.2663, Y 19.5565, Z -3.8333, A 0.000, B 0.000, C 0.000 }
